(* Logix 5000 project; controller WP_Ottawa_Data_Concentrator_1 vendor 1 type 14 code 167 rev 32.14; software revision 32.04 *)
// Data Concentrator

TASK MainTask (continuous, watchdog 500 ms) : MainProgram, LN31

MODULES
   Local : vendor 1 type 14 code 167 (ICP 0, rev 32.14)
      Local_Network : vendor 1 type 12 code 200 (ICP 1, Ethernet 192.168.1.2, rev 11.2)
      Plant_Network : vendor 1 type 12 code 200 (ICP 2, Ethernet 10.31.12.136, rev 11.2)
         WP_Ottawa_Simulator_PLC : vendor 1 type 14 code 156 (Ethernet 10.31.12.137, rev 32.1, $a37dfcfc$ RPI 20 ms)   // WP_Ottawa_Simulator_PLC
         Upr_Line_PLC : vendor 1 type 12 code 200 (Ethernet 10.31.13.135, rev 11.2, Output RPI 10 ms)
            Upright_Line : vendor 1 type 14 code 213 (ICP 0, rev 31.1, $771d54c0$ RPI 20 ms, $aa9c0943$ RPI 20 ms, $f776f99a$ RPI 20 ms, $f5df2af5$ RPI 20 ms, $e50c8bc4$ RPI 20 ms, $a2ad16b7$ RPI 20 ms, $a4c949be$ RPI 20 ms, $f02d2109$ RPI 20 ms, $56660608$ RPI 20 ms, $0d2a626b$ RPI 20 ms, $ec5ac722$ RPI 20 ms, $27c2d75d$ RPI 20 ms, $f8c5678c$ RPI 20 ms, $9b57805f$ RPI 20 ms, $1c2d35c6$ RPI 20 ms, $a70581f1$ RPI 20 ms, $e44b9450$ RPI 20 ms, $3b304493$ RPI 20 ms, $244199aa$ RPI 20 ms, $c2e494c5$ RPI 20 ms, $b4e2b054$ RPI 20 ms, $661cc307$ RPI 20 ms, $eafc36ce$ RPI 20 ms, $ac2dc3d9$ RPI 20 ms)
END_MODULES

TYPE Barcode_SNModel :
STRUCT
   Data : STRING[5];
   Bit : BOOL[32];
END_STRUCT
END_TYPE

TYPE DateTime_Type :   // Structure for the DateTime from the Controller wallclock accessed by the GSV/SSV instruction
STRUCT
   Year : DINT;
   Month : DINT;   // The month (1 - 12)
   Day : DINT;   // The day (1 - 31)
   Hour : DINT;   // hour (0 - 23)
   Minute : DINT;   // minute (0 - 59)
   Second : DINT;   // second (0 - 59)
   Microseconds : DINT;   // (0 - 999,999)
END_STRUCT
END_TYPE

TYPE DC1_To_SIM :
STRUCT
   Status : CONNECTION_STATUS;
   Data : INT[225];
END_STRUCT
END_TYPE

TYPE Line_To_DC :
STRUCT
   Status : CONNECTION_STATUS;
   Data : INT[225];
END_STRUCT
END_TYPE

TYPE PA_WallClock_UDDT :
STRUCT
   One_Shots : BOOL[128];
   Bool : BOOL[128];
   Real : REAL[50];
   Dbl_Int : DINT[50];
   Int : INT[50];
   Pointer1 : INT;
   Pointer2 : INT;
   Pointer3 : INT;
   Pointer4 : INT;
   Pointer5 : INT;
   Timer : TIMER[50];
   Counter : COUNTER[25];
   Control : CONTROL[16];
END_STRUCT
END_TYPE

TYPE SIM_To_DC :
STRUCT
   Status : CONNECTION_STATUS;
   Data : INT[225];
END_STRUCT
END_TYPE

TYPE STRING_12 :
STRUCT
   LEN : DINT;
   DATA : SINT[12];
END_STRUCT
END_TYPE

TYPE STRING_16 :
STRUCT
   LEN : DINT;
   DATA : SINT[16];
END_STRUCT
END_TYPE

TYPE STRING_24 :
STRUCT
   LEN : DINT;
   DATA : SINT[24];
END_STRUCT
END_TYPE

TYPE STRING_4 :
STRUCT
   LEN : DINT;
   DATA : SINT[4];
END_STRUCT
END_TYPE

TYPE STRING_40 :
STRUCT
   LEN : DINT;
   DATA : SINT[40];
END_STRUCT
END_TYPE

TYPE UDT_Current_Status :
STRUCT
   Area : STRING_12;
   Line : STRING_12;
   Shift : DINT;
   _1st_Shift_Avail : BOOL;
   _1st_Shift_Active : BOOL;
   _1st_Shift_Scheduled : BOOL;
   _2nd_Shift_Avail : BOOL;
   _2nd_Shift_Active : BOOL;
   _2nd_Shift_Scheduled : BOOL;
   _3rd_Shift_Avail : BOOL;
   _3rd_Shift_Active : BOOL;
   _3rd_Shift_Scheduled : BOOL;
   DayOfWeek : STRING_16;
   DayOfWeek_Int : DINT;
   Start_Time : STRING_16;
   End_Time : STRING_16;
   _1st_Break_Time : STRING_16;
   _1st_Break_Trigger : BOOL;
   _1st_Break_Active : BOOL;
   _1st_Break_Used : BOOL;
   Lunch_Time : STRING_16;
   Lunch_Trigger : BOOL;
   Lunch_Active : BOOL;
   Lunch_Used : BOOL;
   _2nd_Break_Time : STRING_16;
   _2nd_Break_Trigger : BOOL;
   _2nd_Break_Active : BOOL;
   _2nd_Break_Used : BOOL;
   Rotate_Active : BOOL;
   Rotate_Cmd : BOOL;   // 30 Second Downtime Event to Rotate the Crew
   Scheduled_Units : DINT;
   Line_Rate : DINT;   // Seconds to Construct a Component
   Line_Rate_SP : REAL;
   Units_Remaining : DINT;
   Units_Produced : DINT;
   Units_Scrapped : DINT;
   Units_Lossed : DINT;
   AY_Percent : REAL;
   Shift_Minutes_Remainng : DINT;
   Shift_Seconds_Remaining : DINT;
   DownTime_Code : DINT;
   Flex_Cmd : BOOL;
   Flex_Active : BOOL;
   FlexTo_Line : STRING_16;
   Flex_EndCmd : BOOL;
   Rotate_LEN : REAL;   // seconds
   Brk_LEN : REAL;   // minutes
   Lunch_LEN : REAL;   // minutes
   Break_Stop_On : BOOL;
   Break_Stop_Allowed : BOOL;
   Flex_Stop_On : BOOL;
   Flex_Stop_Allowed : BOOL;
   Rotate_Stop_On : BOOL;
   Rotate_Stop_Allowed : BOOL;
   S1_Scheduled : DINT;
   S2_Scheduled : DINT;
   S3_Scheduled : DINT;
   Shift_Scheduled : BOOL;
   Shift_Active : BOOL;
   RateToMakeSchedule : REAL;
   Theoretical_Units : DINT;
   Standard_LineRate : REAL;
   Running : BOOL;
   State : DINT;
   LineWide_Event : DINT;
   Units_Rejected : DINT;
END_STRUCT
END_TYPE

TYPE UDT_Daily_Schedule :
STRUCT
   _1st_Shift_Avail : BOOL;
   _1st_Shift_Start : STRING_16;
   _1st_Shift_End : STRING_16;
   _1st_Shift_Break1_Start : STRING_16;
   _1st_Shift_Break1_Length : DINT;   // Minutes
   _1st_Shift_Lunch_Start : STRING_16;
   _1st_Shift_Lunch_Length : DINT;   // Minutes
   _1st_Shift_Break2_Start : STRING_16;
   _1st_Shift_Break2_Length : DINT;   // Minutes
   _2nd_Shift_Avail : BOOL;
   _2nd_Shift_Start : STRING_16;
   _2nd_Shift_End : STRING_16;
   _2nd_Shift_Break1_Start : STRING_16;
   _2nd_Shift_Break1_Length : DINT;   // Minutes
   _2nd_Shift_Lunch_Start : STRING_16;
   _2nd_Shift_Lunch_Length : DINT;   // Minutes
   _2nd_Shift_Break2_Start : STRING_16;
   _2nd_Shift_Break2_Length : DINT;   // Minutes
   _3rd_Shift_Avail : BOOL;
   _3rd_Shift_Start : STRING_16;
   _3rd_Shift_End : STRING_16;
   _3rd_Shift_Break1_Start : STRING_16;
   _3rd_Shift_Break1_Length : DINT;   // Minutes
   _3rd_Shift_Lunch_Start : STRING_16;
   _3rd_Shift_Lunch_Length : DINT;   // Minutes
   _3rd_Shift_Break2_Start : STRING_16;
   _3rd_Shift_Break2_Length : DINT;   // Minutes
   Rotate_Length : DINT;   // Seconds
   Break_Stop_On : BOOL;
   Break_Stop_Allowed : BOOL;
   Flex_Stop_On : BOOL;
   Flex_Stop_Allowed : BOOL;
   Rotate_Stop_On : BOOL;
   Rotate_Stop_Allowed : BOOL;
   S1_Scheduled : DINT;
   S2_Scheduled : DINT;
   S3_Scheduled : DINT;
   RateToMakeSchedule : REAL;
END_STRUCT
END_TYPE

TYPE UDT_ShiftString_Breakdown :
STRUCT
   s1StartHour : STRING_4;
   s1StartMin : STRING_4;
   s1EndHour : STRING_4;
   s1_EndMin : STRING_4;
   s2StartHour : STRING_4;
   s2StartMin : STRING_4;
   s2EndHour : STRING_4;
   s2EndMin : STRING_4;
   s3StartHour : STRING_4;
   s3StartMin : STRING_4;
   s3EndHour : STRING_4;
   s3EndMin : STRING_4;
   break1StartHour : STRING_4;
   break1StartMin : STRING_4;
   break2StartHour : STRING_4;
   break2StartMin : STRING_4;
   lunchStartHour : STRING_4;
   lunchStartMin : STRING_4;
END_STRUCT
END_TYPE

TYPE UDT_Weekly_Schedule :
STRUCT
   Monday : UDT_Daily_Schedule;
   Tuesday : UDT_Daily_Schedule;
   Wednesday : UDT_Daily_Schedule;
   Thursday : UDT_Daily_Schedule;
   Friday : UDT_Daily_Schedule;
   Saturday : UDT_Daily_Schedule;
   Sunday : UDT_Daily_Schedule;
END_STRUCT
END_TYPE

VAR_GLOBAL   (* controller tags *)
   ay : REAL := 0.96875;
   clock_current_string : STRING[13] := ([0] := '2023', [1] := '5', [2] := '15', [3] := '14', [4] := '19', [5] := '15');
   Clock_Min_Pulse : BOOL;
   Clock_Set_Routine : PA_WallClock_UDDT := (Dbl_Int[40] := 2023, Dbl_Int[41] := 5, Dbl_Int[42] := 15, Dbl_Int[43] := 14, Dbl_Int[44] := 19, Dbl_Int[45] := 15, Dbl_Int[46] := 696501);
   DateTime_Update : BOOL;
   DayOfWeek : DINT := 1;
   DC1_clock_sync : DINT[10] := ([0] := 2023, [1] := 5, [2] := 15, [3] := 14, [4] := 19, [5] := 12);
   DC1_OPCFault : BOOL := 1;
   DC1_OPCWatchDog : BOOL;
   DC1_To_Line31SIM : DC1_To_SIM := (Status.RunMode := 1, Data[2] := 16); {produced}
   DC1_to_LN31_Messages : DINT[120] := ([2] := 1, [3] := 620, [5] := 20, [6] := 3, [7] := 20, [8] := 3, [9] := 20, [10] := 3, [11] := 20, [12] := 3, [13] := 20, [14] := 3, [15] := 20, [16] := 3, [19] := 1); {produced}
        [10]   // CURRENT SCHEDULE SHIFT 2 START MINUTE
        [11]   // CURRENT SCHEDULE SHIFT 2 END HOUR
        [12]   // CURRENT SCHEDULE SHIFT 2 END MINUTE
        [13]   // CURRENT SCHEDULE SHIFT 3 START HOUR
        [14]   // CURRENT SCHEDULE SHIFT 3 START MINUTE
        [15]   // CURRENT SCHEDULE SHIFT 3 END HOUR
        [16]   // CURRENT SCHEDULE SHIFT 3 END MINUTE
        [19].0   // SHIFT SCHEDULED
        [19].1   // OPC COMMS OKAY
        [19].2   // Shift Reset Timer Complete
        [2]   // ACTIVE SHIFT
        [3]   // Scheduled Units
        [5]   // CURRENT SCHEDULE SHIFT 1 START HOUR
        [6]   // CURRENT SCHEDULE SHIFT 1 START MINUTE
        [7]   // CURRENT SCHEDULE SHIFT 1 END HOUR
        [8]   // CURRENT SCHEDULE SHIFT 1 END MINUTE
        [9]   // CURRENT SCHEDULE SHIFT 2 START HOUR
   fifi_unload : DINT;
   IGN_DateTime_Record_Current : STRING := '2022,09,15,08:55:00';
   IGN_Day : DINT := 15;
   IGN_DayPrev : DINT := 15;
   IGN_DayString : STRING := '15';
   IGN_Hour : DINT := 14;
   IGN_HourString : STRING := '14';
   IGN_Minute : DINT := 19;
   IGN_MinuteString : STRING := '19';
   IGN_Month : DINT := 5;
   IGN_MonthString : STRING := '5';
   IGN_Second : DINT := 10;
   IGN_SecondString : STRING := '12';
   IGN_Year : DINT := 2023;
   IGN_YearString : STRING := '2023';
   Line31SIM_To_DC1 : SIM_To_DC := (Status.RunMode := 1, Data[0] := 12);
   LN31_1st_Station_Break_Code : DINT := 16;
   LN31_Assembly_MNT : DINT;
   LN31_Blocked_At_Run_Test_Exit : DINT;
   LN31_Blocked_By_Penske_CAL : DINT;
   LN31_Blocked_By_Repair : DINT;
   LN31_Blocked_By_Wrapper : DINT;
   LN31_BrazingArea_MNT : DINT;
   LN31_Charge_MNT : DINT;
   LN31_CompressorInstall_MNT : DINT;
   LN31_Current_Shift_Duration_Mins : DINT := 505;
   LN31_Current_Shift_Duration_wBreaks_Mins : DINT := 455;
   LN31_DC_Controlled_Theoretical_Units : BOOL := 1;
   LN31_DowntimeCodesMachineA : DINT[120];
   LN31_DowntimeCodesMachineB : DINT[120];
   LN31_DowntimeCodesMachineC : DINT[120];
   LN31_DowntimeCodesMachineD : DINT[120];
   LN31_DowntimeCodesMachineE : DINT[120];
   LN31_DowntimeCodesMachineF : DINT[120];
   LN31_DowntimeCodesMachineG : DINT[120];
   LN31_DowntimeCodesMachineH : DINT[120];
   LN31_DowntimeCodesMachineI : DINT[120];
   LN31_DowntimeCodesMachineOA : DINT[120];
        [9].0   // LN31 Line Running
        [9].1   // LN31 On Break or Not Scheduled
   LN31_DowntimeCodesMachineX : DINT[120];
   LN31_EStop_HMI1 : DINT;
   LN31_EStop_HMI2 : DINT;
   LN31_EStop_Main_Panel : DINT;
   LN31_EStop_Remote_Panel : DINT;
   LN31_EvacLoop_MNT : DINT;
   LN31_FPY : REAL := 88.08;
   LN31_Ignition_NewSNModel : BOOL[32];
   LN31_Ignition_SNModelMSG : STRING[5] := ([0] := 'WZF34X18DW 07', [1] := 'UC2001942');
   LN31_InspectionAndTest_MNT : DINT;
   LN31_Kit_Zone_1_Exit_Fault : DINT;
   LN31_Kitting_MNT : DINT;
   LN31_Label_Machines_Faulted : DINT;
   LN31_Label_Missing : DINT;
   LN31_MachineOverAll_MNT : DINT;
   LN31_Messages_Barcode_SNModel : Barcode_SNModel := (Data[0] := 'WZF34X18DW 07', Data[1] := 'UC2001942');
   LN31_Miscellaneous_MNT : DINT;
   LN31_MLC_Downtime : BOOL;
   LN31_Packout_MNT : DINT;
   LN31_PrefoamGlueAndFoam_MNT : DINT;
   LN31_Schedule : UDT_Current_Status := (Line := 'LN31', Shift := 1, _1st_Shift_Avail := 1, _1st_Shift_Active := 1, _1st_Shift_Scheduled := 1, _3rd_Shift_Scheduled := 1, DayOfWeek := 'Mon', DayOfWeek_Int := 1, Start_Time := '2023-05-15 07:05', End_Time := '2023-05-15 15:30', _1st_Break_Time := '09:10', Lunch_Time := '12:10', _2nd_Break_Time := '20:30', Scheduled_Units := 620, Line_Rate := 56, Units_Remaining := 415, Units_Produced := 411, Units_Lossed := 13, AY_Percent := 96.875, Break_Stop_Allowed := 1, Shift_Scheduled := 1, Shift_Active := 1, Theoretical_Units := 522, Running := 1, State := 3, Units_Rejected := 49);
        .Units_Lossed   // LN31 Rejected Count
   LN31_Schedule_Cycle_Timer : TIMER := (PRE := 44032, ACC := 751, EN := 1, TT := 1);
   LN31_Schedule_Max_Break_Duration : DINT := 50;
   LN31_Schedule_Max_Break_Timer : TIMER := (PRE := 3000000, ACC := 3000000, EN := 1, DN := 1);
   LN31_Schedule_TAKT : REAL := 44032.258;
   LN31_Scheduled_Units_Buffer : DINT := 620;
   LN31_ScheduleUnits_Produced_from_line : DINT := 412;
   LN31_Starved_By_Surge : DINT;
   LN31_Surge_Gate_Open : DINT;
   LN31_Theoretical_Units_Counter : COUNTER := (PRE := 999999, ACC := 522);
   LN31_Theoretical_Units_Counter_ONS : BOOL;
   LN31_to_DC01_Main_Messages : Line_To_DC := (Status.RunMode := 1, Data[4] := 543, Data[6] := 44, Data[9] := 1, Data[15] := 8637, Data[18] := 618, Data[19] := 74);
   LN31_Toggle_CountSource : BOOL;
   LN31_Weekly_Schedule : UDT_Weekly_Schedule := (Monday._1st_Shift_Avail := 1, Monday._1st_Shift_Start := '2023-05-15 07:05', Monday._1st_Shift_End := '2023-05-15 15:30', Monday._1st_Shift_Break1_Start := '09:10', Monday._1st_Shift_Break1_Length := 15, Monday._1st_Shift_Lunch_Start := '12:10', Monday._1st_Shift_Lunch_Length := 30, Monday._1st_Shift_Break2_Start := '20:30', Monday._1st_Shift_Break2_Length := 15, Monday._2nd_Shift_Start := '2023-05-15 20:25', Monday._2nd_Shift_End := '2023-05-15 20:30', Monday._2nd_Shift_Break1_Start := '17:45', Monday._2nd_Shift_Break1_Length := 15, Monday._2nd_Shift_Lunch_Start := '20:30', Monday._2nd_Shift_Lunch_Length := 30, Monday._2nd_Shift_Break2_Start := '12:10', Monday._2nd_Shift_Break2_Length := 15, Monday._3rd_Shift_Avail := 1, Monday._3rd_Shift_Start := '2023-05-14 21:35', Monday._3rd_Shift_End := '2023-05-15 06:00', Monday._3rd_Shift_Break1_Start := '01:00', Monday._3rd_Shift_Break1_Length := 15, Monday._3rd_Shift_Lunch_Start := '03:00', Monday._3rd_Shift_Lunch_Length := 30, Monday._3rd_Shift_Break2_Start := '04:00', Monday._3rd_Shift_Break2_Length := 15, Monday.S1_Scheduled := 620, Monday.S3_Scheduled := 620, Tuesday._1st_Shift_Avail := 1, Tuesday._1st_Shift_Start := '2023-05-16 07:05', Tuesday._1st_Shift_End := '2023-05-16 15:30', Tuesday._1st_Shift_Break1_Start := '09:10', Tuesday._1st_Shift_Break1_Length := 15, Tuesday._1st_Shift_Lunch_Start := '12:10', Tuesday._1st_Shift_Lunch_Length := 30, Tuesday._1st_Shift_Break2_Start := '20:30', Tuesday._1st_Shift_Break2_Length := 15, Tuesday._2nd_Shift_Start := '2023-05-16 20:25', Tuesday._2nd_Shift_End := '2023-05-16 20:30', Tuesday._2nd_Shift_Break1_Start := '17:45', Tuesday._2nd_Shift_Break1_Length := 15, Tuesday._2nd_Shift_Lunch_Start := '20:30', Tuesday._2nd_Shift_Lunch_Length := 30, Tuesday._2nd_Shift_Break2_Start := '12:10', Tuesday._2nd_Shift_Break2_Length := 15, Tuesday._3rd_Shift_Avail := 1, Tuesday._3rd_Shift_Start := '2023-05-15 21:35', Tuesday._3rd_Shift_End := '2023-05-16 06:00', Tuesday._3rd_Shift_Break1_Start := '1:00', Tuesday._3rd_Shift_Break1_Length := 15, Tuesday._3rd_Shift_Lunch_Start := '03:00', Tuesday._3rd_Shift_Lunch_Length := 30, Tuesday._3rd_Shift_Break2_Start := '04:00', Tuesday._3rd_Shift_Break2_Length := 15, Tuesday.S1_Scheduled := 620, Tuesday.S3_Scheduled := 620, Wednesday._1st_Shift_Avail := 1, Wednesday._1st_Shift_Start := '2023-05-17 07:05', Wednesday._1st_Shift_End := '2023-05-17 15:30', Wednesday._1st_Shift_Break1_Start := '09:10',
        Wednesday._1st_Shift_Break1_Length := 15, Wednesday._1st_Shift_Lunch_Start := '12:10', Wednesday._1st_Shift_Lunch_Length := 30, Wednesday._1st_Shift_Break2_Start := '20:30', Wednesday._1st_Shift_Break2_Length := 15, Wednesday._2nd_Shift_Start := '2023-05-17 20:25', Wednesday._2nd_Shift_End := '2023-05-17 20:30', Wednesday._2nd_Shift_Break1_Start := '17:45', Wednesday._2nd_Shift_Break1_Length := 15, Wednesday._2nd_Shift_Lunch_Start := '20:30', Wednesday._2nd_Shift_Lunch_Length := 30, Wednesday._2nd_Shift_Break2_Start := '12:10', Wednesday._2nd_Shift_Break2_Length := 15, Wednesday._3rd_Shift_Avail := 1, Wednesday._3rd_Shift_Start := '2023-05-16 21:35', Wednesday._3rd_Shift_End := '2023-05-17 06:00', Wednesday._3rd_Shift_Break1_Start := '01:00', Wednesday._3rd_Shift_Break1_Length := 15, Wednesday._3rd_Shift_Lunch_Start := '03:00', Wednesday._3rd_Shift_Lunch_Length := 30, Wednesday._3rd_Shift_Break2_Start := '04:00', Wednesday._3rd_Shift_Break2_Length := 15, Wednesday.S1_Scheduled := 620, Wednesday.S3_Scheduled := 620, Thursday._1st_Shift_Avail := 1, Thursday._1st_Shift_Start := '2023-05-18 07:05', Thursday._1st_Shift_End := '2023-05-18 15:30', Thursday._1st_Shift_Break1_Start := '09:10', Thursday._1st_Shift_Break1_Length := 15, Thursday._1st_Shift_Lunch_Start := '12:10', Thursday._1st_Shift_Lunch_Length := 30, Thursday._1st_Shift_Break2_Start := '20:30', Thursday._1st_Shift_Break2_Length := 15, Thursday._2nd_Shift_Start := '2023-05-18 20:25', Thursday._2nd_Shift_End := '2023-05-18 20:30', Thursday._2nd_Shift_Break1_Start := '17:45', Thursday._2nd_Shift_Break1_Length := 15, Thursday._2nd_Shift_Lunch_Start := '20:30', Thursday._2nd_Shift_Lunch_Length := 30, Thursday._2nd_Shift_Break2_Start := '12:10', Thursday._2nd_Shift_Break2_Length := 15, Thursday._3rd_Shift_Avail := 1, Thursday._3rd_Shift_Start := '2023-05-17 21:35', Thursday._3rd_Shift_End := '2023-05-18 06:00', Thursday._3rd_Shift_Break1_Start := '01:00', Thursday._3rd_Shift_Break1_Length := 15, Thursday._3rd_Shift_Lunch_Start := '03:00', Thursday._3rd_Shift_Lunch_Length := 30, Thursday._3rd_Shift_Break2_Start := '04:00', Thursday._3rd_Shift_Break2_Length := 15, Thursday.S1_Scheduled := 620, Thursday.S3_Scheduled := 620, Friday._1st_Shift_Avail := 1, Friday._1st_Shift_Start := '2023-05-19 07:05', Friday._1st_Shift_End := '2023-05-19 15:30', Friday._1st_Shift_Break1_Start := '09:10', Friday._1st_Shift_Break1_Length := 15, Friday._1st_Shift_Lunch_Start := '12:10', Friday._1st_Shift_Lunch_Length := 30, Friday._1st_Shift_Break2_Start := '20:30',
        Friday._1st_Shift_Break2_Length := 15, Friday._2nd_Shift_Start := '2023-05-19 20:25', Friday._2nd_Shift_End := '2023-05-19 20:30', Friday._2nd_Shift_Break1_Start := '17:45', Friday._2nd_Shift_Break1_Length := 15, Friday._2nd_Shift_Lunch_Start := '20:30', Friday._2nd_Shift_Lunch_Length := 30, Friday._2nd_Shift_Break2_Start := '12:10', Friday._2nd_Shift_Break2_Length := 15, Friday._3rd_Shift_Avail := 1, Friday._3rd_Shift_Start := '2023-05-18 21:35', Friday._3rd_Shift_End := '2023-05-19 06:00', Friday._3rd_Shift_Break1_Start := '01:00', Friday._3rd_Shift_Break1_Length := 15, Friday._3rd_Shift_Lunch_Start := '03:00', Friday._3rd_Shift_Lunch_Length := 30, Friday._3rd_Shift_Break2_Start := '04:00', Friday._3rd_Shift_Break2_Length := 15, Friday.S1_Scheduled := 620, Friday.S3_Scheduled := 620, Saturday._1st_Shift_Start := '2023-05-20 07:05', Saturday._1st_Shift_End := '2023-05-20 16:30', Saturday._1st_Shift_Break1_Start := '09:10', Saturday._1st_Shift_Break1_Length := 15, Saturday._1st_Shift_Lunch_Start := '12:10', Saturday._1st_Shift_Lunch_Length := 30, Saturday._1st_Shift_Break2_Start := '18:45', Saturday._1st_Shift_Break2_Length := 15, Saturday._2nd_Shift_Start := '2023-05-20 17:00', Saturday._2nd_Shift_End := '2023-05-20 17:01', Saturday._2nd_Shift_Break1_Start := '17:45', Saturday._2nd_Shift_Break1_Length := 15, Saturday._2nd_Shift_Lunch_Start := '20:30', Saturday._2nd_Shift_Lunch_Length := 30, Saturday._2nd_Shift_Break2_Start := '12:10', Saturday._2nd_Shift_Break2_Length := 15, Saturday._3rd_Shift_Start := '2023-05-19 20:35', Saturday._3rd_Shift_End := '2023-05-20 06:00', Saturday._3rd_Shift_Break1_Start := '01:00', Saturday._3rd_Shift_Break1_Length := 15, Saturday._3rd_Shift_Lunch_Start := '03:00', Saturday._3rd_Shift_Lunch_Length := 30, Saturday._3rd_Shift_Break2_Start := '05:00', Saturday._3rd_Shift_Break2_Length := 15, Sunday._1st_Shift_Start := '2023-05-21 07:05', Sunday._1st_Shift_End := '2023-05-21 16:30', Sunday._1st_Shift_Break1_Start := '09:0', Sunday._1st_Shift_Break1_Length := 15, Sunday._1st_Shift_Lunch_Start := '12:10', Sunday._1st_Shift_Lunch_Length := 30, Sunday._1st_Shift_Break2_Start := '18:45', Sunday._1st_Shift_Break2_Length := 15, Sunday._2nd_Shift_Start := '2023-05-21 17:00', Sunday._2nd_Shift_End := '2023-05-21 17:01', Sunday._2nd_Shift_Break1_Start := '17:45', Sunday._2nd_Shift_Break1_Length := 30, Sunday._2nd_Shift_Lunch_Start := '20:30', Sunday._2nd_Shift_Lunch_Length := 30, Sunday._2nd_Shift_Break2_Start := '12:10', Sunday._2nd_Shift_Break2_Length := 15,
        Sunday._3rd_Shift_Start := '2023-05-20 20:35', Sunday._3rd_Shift_End := '2023-05-21 06:00', Sunday._3rd_Shift_Break1_Start := '01:00', Sunday._3rd_Shift_Break1_Length := 140, Sunday._3rd_Shift_Lunch_Start := '03:00', Sunday._3rd_Shift_Lunch_Length := 30, Sunday._3rd_Shift_Break2_Start := '05:00', Sunday._3rd_Shift_Break2_Length := 10);
   LN31_WorkstationsA : DINT[120];
   LN31_WorkstationsB : DINT[120] := ([3] := 1048592);
   LN31_WorkstationsC : DINT[120];
   LN31_WorkstationsD : DINT[120];
   LN31_WorkstationsE : DINT[120];
   LN31_WorkstationsF : DINT[120];
   LN31_WorkstationsG : DINT[120];
   LN31_WorkstationsH : DINT[120];
   LN31_WorkstationsI : DINT[120];
   LN31_WorkstationsOA : DINT[120] := ([4] := 411, [6] := 56, [9] := 1, [15] := 8808, [16] := 49, [17] := 1, [18] := 410);
        [15]   // LN31 Lodestar FPY Decimal as Integer
        [17]   // LN31 Active Shift
        [18]   // LN31 Scheduled Units (Run Target Count)
        [19]   // LN31 Lost Unit Count ( Reject Count)
        [20]   // LN31 Main Line Active DT Code
        [21]   // LN31 Sub Process 1 Machine DT Code
        [22]   // LN31 Sub Process 2 Machine DT Code
        [23]   // LN31 Sub Process 3 Machine DT Code
        [24]   // LN31 Sub Process 4 Machine DT Code
        [25]   // LN31 Sub Process 5 Machine DT Code
        [26]   // LN31 Sub Process 6 Machine DT Code
        [27]   // LN31 Sub Process 7 Machine DT Code
        [28]   // LN31 Sub Process 8 Machine DT Code
        [29]   // LN31 Sub Process 9 Machine DT Code
        [30]   // LN31 Sub Process 10 Machine DT Code
        [4]   // LN31 Actual Unit Count (Lodestar Crated)
        [6]   // LN31 Takt Target Time
        [9].0   // Line Running
        [9].1   // On Break or Not Scheduled
   LN31_WorkstationsX : DINT[120] := ([7] := 1048592, [8] := 1048592, [9] := 1048592, [10] := 1048592, [11] := 1048592, [12] := 1048592);
   LN31_Wrong_Compressor : DINT;
   LN31_Z22F_Over_Cycle_Time : DINT;
   LN31EAM02 : DINT;
   LN31EAM03 : DINT;
   LN31EFM01 : DINT;
   LN31EFM02 : DINT;
   LN31EFM03 : DINT;
   LN31EGM01 : DINT;
   LN31EGM02 : DINT;
   LN31EGM03 : DINT;
   LN31EGM04 : DINT;
   LN31EHS01 : DINT;
   LN31EHS02 : DINT;
   LN31EHS03 : DINT;
   LN31EHS04 : DINT;
   LN31EHS05 : DINT;
   LN31EHS06 : DINT;
   LN31EHS07 : DINT;
   LN31EHS08 : DINT;
   LN31EIS05 : DINT;
   LN31NCM02 : DINT;
   LN31NDM01 : DINT;
   LN31NDM02 : DINT;
   LN31NDM03 : DINT;
   LN31NIS02 : DINT;
   LN31NIS03 : DINT;
   LN31NIS04 : DINT;
   LN31NIS06 : DINT;
   LN31NIS07 : DINT;
   LN31NIS08 : DINT;
   LN31NIS09 : DINT;
   LN31NIS10 : DINT;
   LN31NIS11 : DINT;
   LN31NIS12 : DINT;
   LN31NIS13 : DINT;
   LN31NIS14 : DINT;
   LN31NIS15 : DINT;
   LN31NIS16 : DINT;
   LN31NIS17 : DINT;
   LN31SBM01 : DINT;
   LN31SBM02 : DINT;
   LN31SBM03 : DINT;
   LN31SBM04 : DINT;
   LN31SBM05 : DINT;
   LN31SCM01 : DINT;
   LN31SDM03 : DINT;
   LN31SIS02 : DINT;
   LN31SIS06 : DINT;
   LN31WAM01 : DINT;
   LN31WAM02 : DINT;
   LN31WEM01 : DINT;
   LN31WEM02 : DINT;
   LN31WEM03 : DINT;
   LN31WEM04 : DINT;
   LN31WEM05 : DINT;
   LN31WEM06 : DINT;
   LN31WEM07 : DINT;
   LN31WEM08 : DINT;
   LN31WEM09 : DINT;
   LN31WFM01 : DINT;
   LN31WFM02 : DINT;
   LN31WFM03 : DINT;
   LN31WGM02 : DINT;
   LN31WGM04 : DINT;
   LN31WIS01 : DINT;
   LN31XAM01 : DINT;
   LN31XAM02 : DINT;
   LN31XAS01 : DINT;
   LN31XAS02 : DINT;
   LN31XBM01 : DINT;
   LN31XBM02 : DINT;
   LN31XBS01 : DINT;
   LN31XBS02 : DINT;
   LN31XCM01 : DINT;
   LN31XCM02 : DINT;
   LN31XCS01 : DINT;
   LN31XCS02 : DINT;
   LN31XDM01 : DINT;
   LN31XDM02 : DINT;
   LN31XDS01 : DINT;
   LN31XDS02 : DINT;
   LN31XEM01 : DINT;
   LN31XEM02 : DINT;
   LN31XES01 : DINT;
   LN31XES02 : DINT;
   LN31XFM01 : DINT;
   LN31XFM02 : DINT;
   LN31XFS01 : DINT;
   LN31XFS02 : DINT;
   LN31XGM01 : DINT;
   LN31XGM02 : DINT;
   LN31XGS01 : DINT;
   LN31XGS02 : DINT;
   LN31XHM01 : DINT;
   LN31XHM02 : DINT;
   LN31XHS01 : DINT;
   LN31XHS02 : DINT;
   LN31XIM01 : DINT;
   LN31XIM02 : DINT;
   LN31XIM03 : DINT;
   LN31XIS01 : DINT;
   LN31XIS02 : DINT;
   LN31XIS03 : DINT;
   local : TIMER := (PRE := 2000, ACC := 1827, EN := 1, TT := 1);
   null : STRING;
   NULL_String : STRING;
   Previous_Shift_Count : DINT := 463;
   scc : CONTROL := (LEN := 60, POS := 59);   // Shift Count History
   Shift_count_history : DINT[62];
   Shift_reset_timer : TIMER := (PRE := 2000);
   Test : MESSAGE;
        MessageParameters(ServiceCode := 16#004c, LocalElement := Test1, ...)
   Test1 : DINT;
   Test_Result : DINT := 1;
   TestDateTime : DINT;
   THEORETICAL_TEST : BOOL;
END_VAR

PROGRAM LN31   (* main routine MainRoutine *)
VAR
   Average_Array : DINT[20] := ([0] := 30000, [1] := 30000, [2] := 30000, [3] := 30000, [4] := 30000, [5] := 30000, [6] := 30000, [7] := 30000, [8] := 30000, [9] := 30000);   // AVERAGE UNIT ASSEMBLY TIME (LAST 10 UNITS)
   Average_Sum : DINT := 300000;
   Averaged_LineSpeed : REAL := 30.0;
   badModel : STRING_40;
   Break1_Hour : DINT := 9;
   Break1_Hour_String : STRING_4 := '09';
   Break1_Length : DINT := 15;
   Break1_Min : DINT := 10;
   Break1_Min_String : STRING_4 := '10';
   Break2_Hour : DINT := 20;
   Break2_Hour_String : STRING_4 := '20';
   Break2_Length : DINT := 15;
   Break2_Min : DINT := 30;
   Break2_Min_String : STRING_4 := '30';
   Break_1stStation : BOOL;
   Break_LineWide : BOOL;
   Break_WorkCenter : BOOL;
   Break_Workstation : BOOL;
   CurrentSchedule : UDT_ShiftString_Breakdown := (s1StartHour := '20', s1StartMin := '3-', s1EndHour := '20', s1_EndMin := '3-', s2StartHour := '20', s2StartMin := '3-', s2EndHour := '20', s2EndMin := '3-', s3StartHour := '20', s3StartMin := '3-', s3EndHour := '20', s3EndMin := '3-');
   End_Hour : DINT := 20;
   End_Hour_String : STRING_4 := '20';
   End_Min : DINT := 3;
   End_Min_String : STRING_4 := '3-';
   firstCharacter : STRING_40 := 'W';
   Local_Timer : TIMER[10] := ([0].PRE := 30000, [0].ACC := 30000, [0].EN := 1, [0].DN := 1, [1].PRE := 4000, [1].ACC := 4000, [1].EN := 1, [1].DN := 1, [2].PRE := 8000, [3].PRE := 2000, [3].ACC := 1538, [3].EN := 1, [3].TT := 1, [4].PRE := 280, [4].ACC := 95, [4].EN := 1, [4].TT := 1);
        [0]   // UNIT ASSEMBLY TIMER
        [1]   // BARCODE TRANSFER TO LODESTAR TRIGGER TIMER
        [2]   // BARCOE TRANFER TO LODESTAR SECOND CHANCE TIMER
        [3]   // LINE PLC WRITE MESSAGE INSTRUCTION TIMER
        [4]   // LINE PLC READ MESSAGE INSTRUCTION TIMER
   Lunch_Hour : DINT := 12;
   Lunch_Hour_String : STRING_4 := '12';
   Lunch_Length : DINT := 30;
   Lunch_Min : DINT := 10;
   Lunch_Min_String : STRING_4 := '10';
   msg192_reset_timer : TIMER := (PRE := 3000);
   ONS_20 : DINT := 3;
        .0   // BARCODE READ FROM LODESTAR STATUS ONE SHOT
        .1   // CLEAR BARCODE READ FROM LODESTAR STATUS ONE SHOT
   PreviousCount : DINT := 411;
   previousSerialNumber : STRING := 'M91940611';
   PreviousShift : DINT := 1;
   readIndex : DINT := 31;
   register : DINT := 9;   // ARRAY POINTER FOR AVERAGE ASSEMBLY TIME ARRAY
   Shift_Reset : BOOL;
   Shift_Reset_ONS : BOOL := 1;
   Start_Hour : DINT := 20;
   Start_Hour_String : STRING_4 := '20';
   Start_Min : DINT := 3;
   Start_Min_String : STRING_4 := '3-';
   tempIndex : DINT := 22;
   theoreticalUnitsReal : REAL;
   writeIndex : DINT;
END_VAR

ROUTINE MainRoutine   (* ladder *)
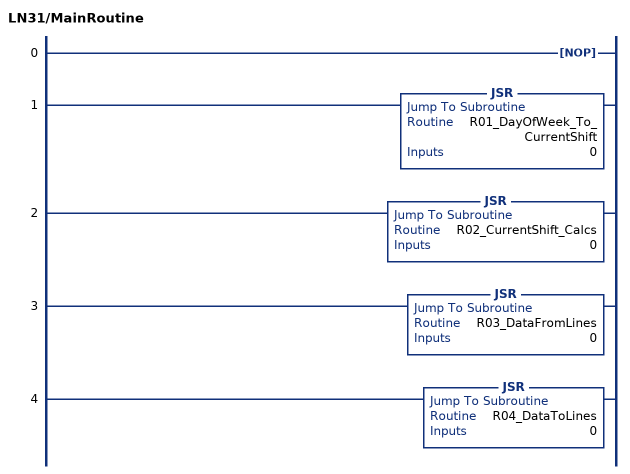
   0: NOP();
   1: JSR(R01_DayOfWeek_To_CurrentShift,0);
   2: JSR(R02_CurrentShift_Calcs,0);
   3: JSR(R03_DataFromLines,0);
   4: JSR(R04_DataToLines,0);
END_ROUTINE

ROUTINE R01_DayOfWeek_To_CurrentShift   (* ladder *)
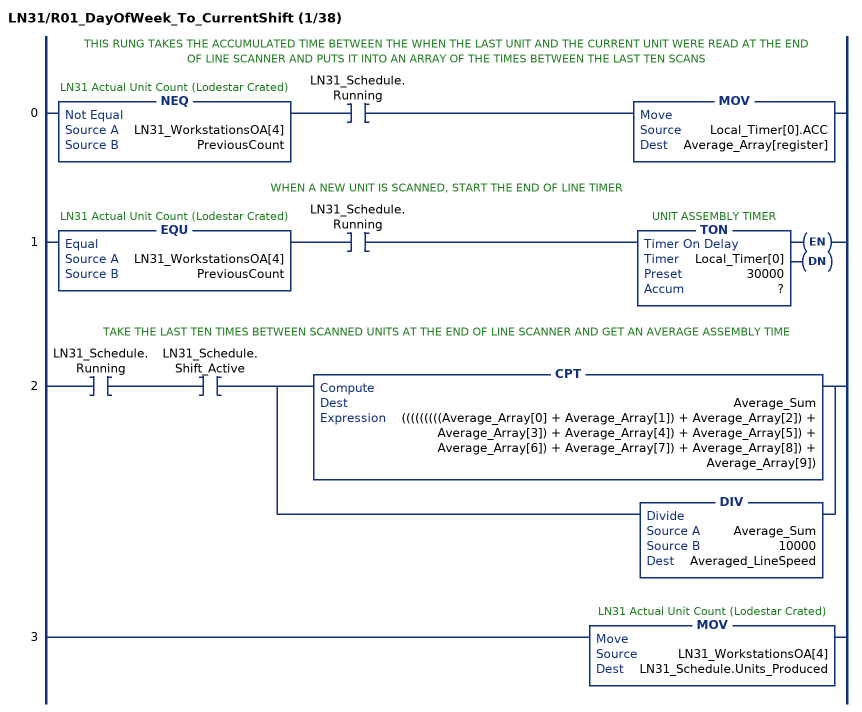
   // THIS RUNG TAKES THE ACCUMULATED TIME BETWEEN THE WHEN THE LAST UNIT AND THE CURRENT UNIT WERE READ AT THE END OF LINE SCANNER AND PUTS IT INTO AN ARRAY OF THE TIMES BETWEEN THE LAST TEN SCANS
   0: NEQ(LN31_WorkstationsOA[4],PreviousCount)XIC(LN31_Schedule.Running)MOV(Local_Timer[0].ACC,Average_Array[register]);
   // WHEN A NEW UNIT IS SCANNED, START THE END OF LINE TIMER
   1: EQU(LN31_WorkstationsOA[4],PreviousCount)XIC(LN31_Schedule.Running)TON(Local_Timer[0],?,?);
   // TAKE THE LAST TEN TIMES BETWEEN SCANNED UNITS AT THE END OF LINE SCANNER AND GET AN AVERAGE ASSEMBLY TIME
   2: XIC(LN31_Schedule.Running)XIC(LN31_Schedule.Shift_Active)[CPT(Average_Sum,(((((((((Average_Array[0] + Average_Array[1]) + Average_Array[2]) + Average_Array[3]) + Average_Array[4]) + Average_Array[5]) + Average_Array[6]) + Average_Array[7]) + Average_Array[8]) + Average_Array[9])) ,DIV(Average_Sum,10000,Averaged_LineSpeed) ];
   3: MOV(LN31_WorkstationsOA[4],LN31_Schedule.Units_Produced);
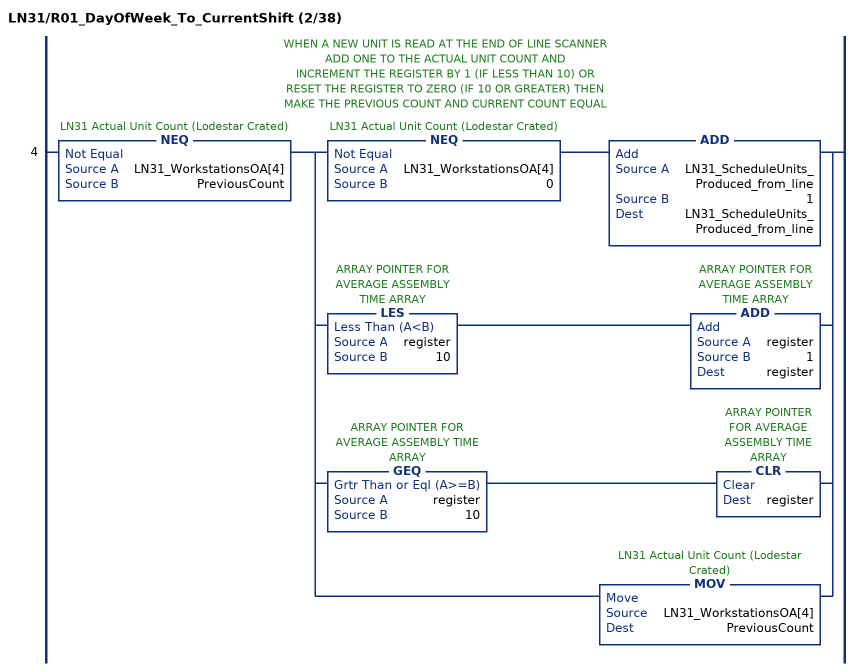
   // WHEN A NEW UNIT IS READ AT THE END OF LINE SCANNER
   // ADD ONE TO THE ACTUAL UNIT COUNT AND
   // INCREMENT THE REGISTER BY 1 (IF LESS THAN 10) OR
   // RESET THE REGISTER TO ZERO (IF 10 OR GREATER) THEN
   // MAKE THE PREVIOUS COUNT AND CURRENT COUNT EQUAL
   4: NEQ(LN31_WorkstationsOA[4],PreviousCount)[NEQ(LN31_WorkstationsOA[4],0) ADD(LN31_ScheduleUnits_Produced_from_line,1,LN31_ScheduleUnits_Produced_from_line) ,LES(register,10) ADD(register,1,register) ,GEQ(register,10) CLR(register) ,MOV(LN31_WorkstationsOA[4],PreviousCount) ];
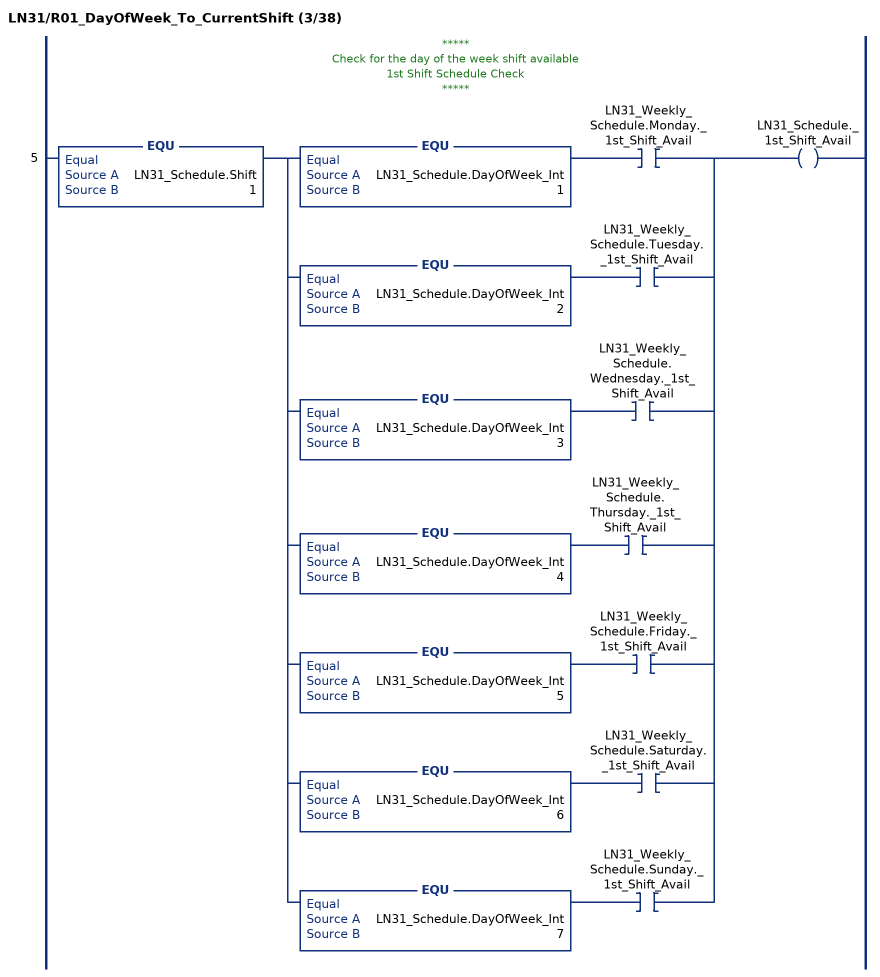
   // *****
   // Check for the day of the week shift available
   // 1st Shift Schedule Check
   // *****
   5: EQU(LN31_Schedule.Shift,1)[EQU(LN31_Schedule.DayOfWeek_Int,1) XIC(LN31_Weekly_Schedule.Monday._1st_Shift_Avail) ,EQU(LN31_Schedule.DayOfWeek_Int,2) XIC(LN31_Weekly_Schedule.Tuesday._1st_Shift_Avail) ,EQU(LN31_Schedule.DayOfWeek_Int,3) XIC(LN31_Weekly_Schedule.Wednesday._1st_Shift_Avail) ,EQU(LN31_Schedule.DayOfWeek_Int,4) XIC(LN31_Weekly_Schedule.Thursday._1st_Shift_Avail) ,EQU(LN31_Schedule.DayOfWeek_Int,5) XIC(LN31_Weekly_Schedule.Friday._1st_Shift_Avail) ,EQU(LN31_Schedule.DayOfWeek_Int,6) XIC(LN31_Weekly_Schedule.Saturday._1st_Shift_Avail) ,EQU(LN31_Schedule.DayOfWeek_Int,7) XIC(LN31_Weekly_Schedule.Sunday._1st_Shift_Avail) ]OTE(LN31_Schedule._1st_Shift_Avail);
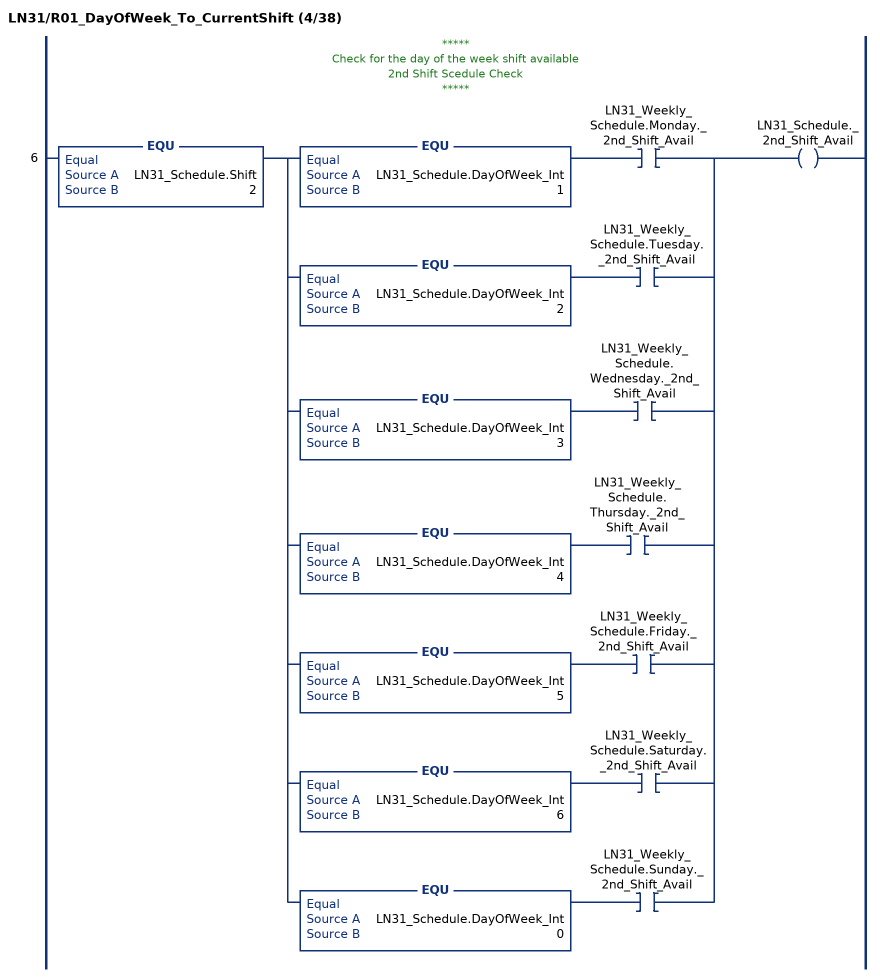
   // *****
   // Check for the day of the week shift available
   // 2nd Shift Scedule Check
   // *****
   6: EQU(LN31_Schedule.Shift,2)[EQU(LN31_Schedule.DayOfWeek_Int,1) XIC(LN31_Weekly_Schedule.Monday._2nd_Shift_Avail) ,EQU(LN31_Schedule.DayOfWeek_Int,2) XIC(LN31_Weekly_Schedule.Tuesday._2nd_Shift_Avail) ,EQU(LN31_Schedule.DayOfWeek_Int,3) XIC(LN31_Weekly_Schedule.Wednesday._2nd_Shift_Avail) ,EQU(LN31_Schedule.DayOfWeek_Int,4) XIC(LN31_Weekly_Schedule.Thursday._2nd_Shift_Avail) ,EQU(LN31_Schedule.DayOfWeek_Int,5) XIC(LN31_Weekly_Schedule.Friday._2nd_Shift_Avail) ,EQU(LN31_Schedule.DayOfWeek_Int,6) XIC(LN31_Weekly_Schedule.Saturday._2nd_Shift_Avail) ,EQU(LN31_Schedule.DayOfWeek_Int,0) XIC(LN31_Weekly_Schedule.Sunday._2nd_Shift_Avail) ]OTE(LN31_Schedule._2nd_Shift_Avail);
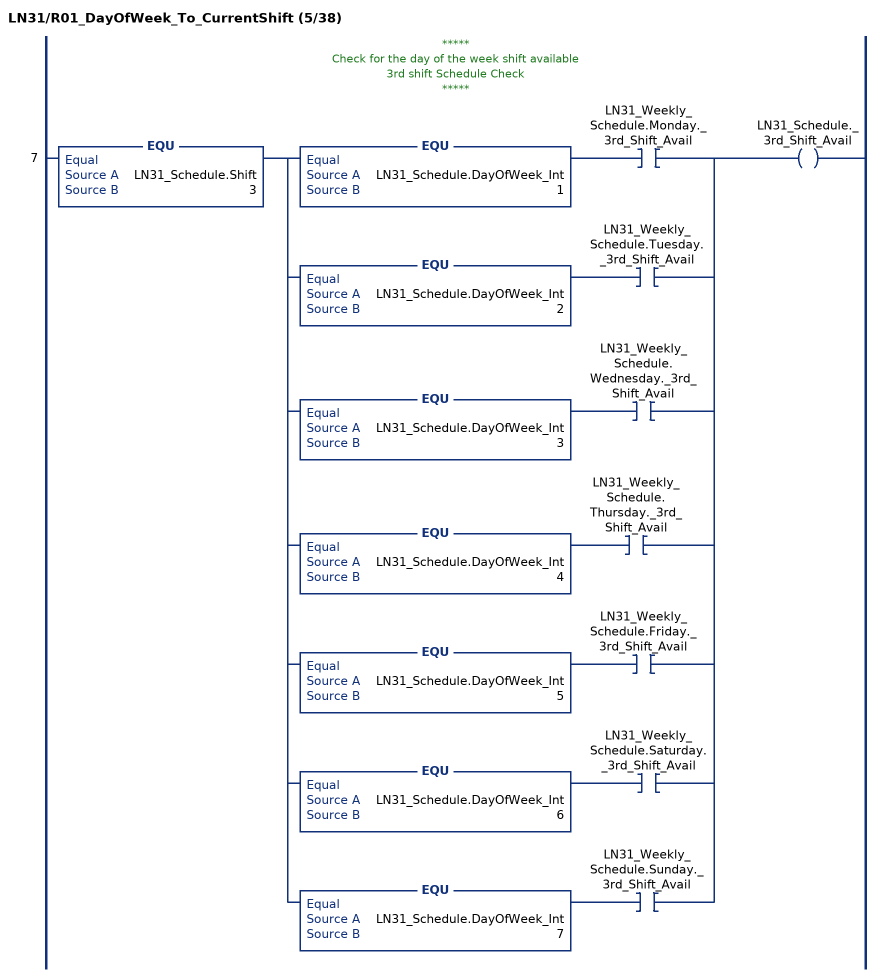
   // *****
   // Check for the day of the week shift available
   // 3rd shift Schedule Check
   // *****
   7: EQU(LN31_Schedule.Shift,3)[EQU(LN31_Schedule.DayOfWeek_Int,1) XIC(LN31_Weekly_Schedule.Monday._3rd_Shift_Avail) ,EQU(LN31_Schedule.DayOfWeek_Int,2) XIC(LN31_Weekly_Schedule.Tuesday._3rd_Shift_Avail) ,EQU(LN31_Schedule.DayOfWeek_Int,3) XIC(LN31_Weekly_Schedule.Wednesday._3rd_Shift_Avail) ,EQU(LN31_Schedule.DayOfWeek_Int,4) XIC(LN31_Weekly_Schedule.Thursday._3rd_Shift_Avail) ,EQU(LN31_Schedule.DayOfWeek_Int,5) XIC(LN31_Weekly_Schedule.Friday._3rd_Shift_Avail) ,EQU(LN31_Schedule.DayOfWeek_Int,6) XIC(LN31_Weekly_Schedule.Saturday._3rd_Shift_Avail) ,EQU(LN31_Schedule.DayOfWeek_Int,7) XIC(LN31_Weekly_Schedule.Sunday._3rd_Shift_Avail) ]OTE(LN31_Schedule._3rd_Shift_Avail);
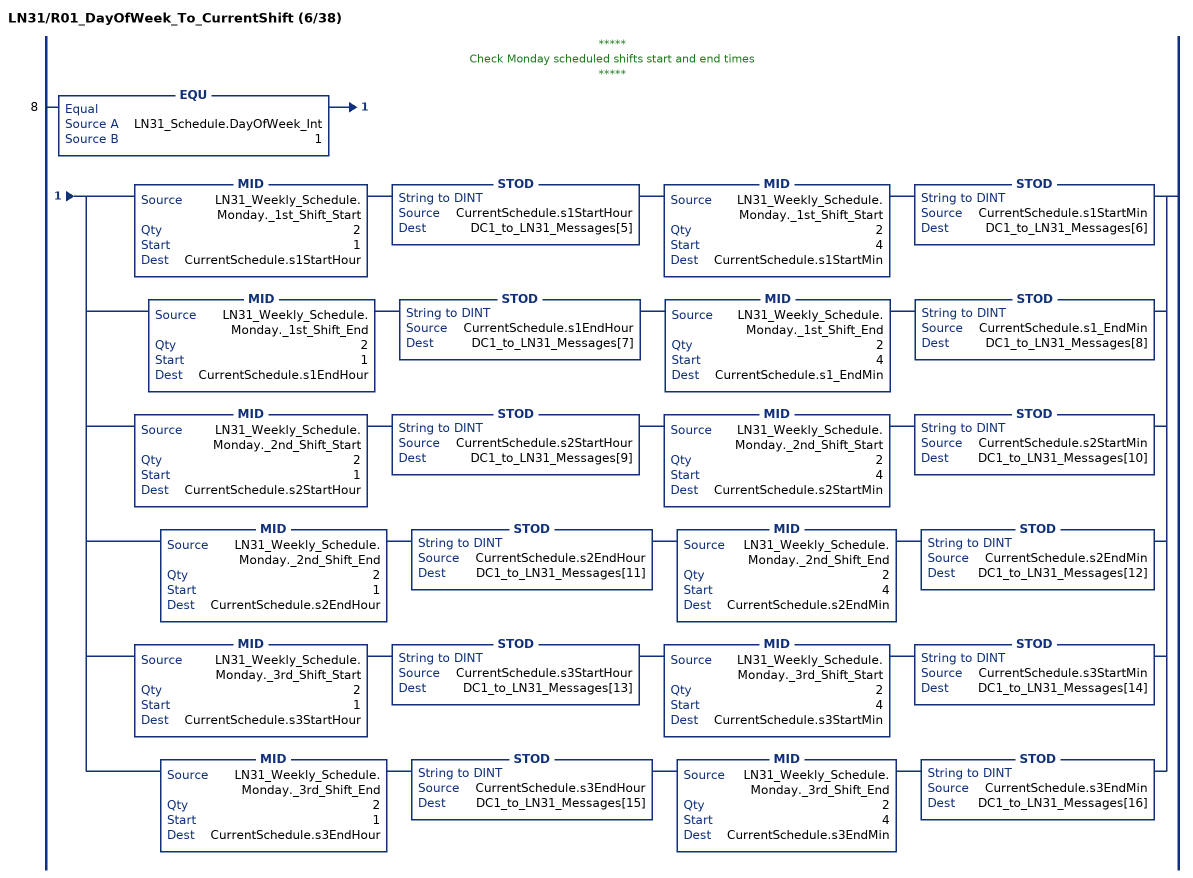
   // *****
   // Check Monday scheduled shifts start and end times
   // *****
   8: EQU(LN31_Schedule.DayOfWeek_Int,1)[MID(LN31_Weekly_Schedule.Monday._1st_Shift_Start,2,1,CurrentSchedule.s1StartHour) STOD(CurrentSchedule.s1StartHour,DC1_to_LN31_Messages[5]) MID(LN31_Weekly_Schedule.Monday._1st_Shift_Start,2,4,CurrentSchedule.s1StartMin) STOD(CurrentSchedule.s1StartMin,DC1_to_LN31_Messages[6]) ,MID(LN31_Weekly_Schedule.Monday._1st_Shift_End,2,1,CurrentSchedule.s1EndHour) STOD(CurrentSchedule.s1EndHour,DC1_to_LN31_Messages[7]) MID(LN31_Weekly_Schedule.Monday._1st_Shift_End,2,4,CurrentSchedule.s1_EndMin) STOD(CurrentSchedule.s1_EndMin,DC1_to_LN31_Messages[8]) ,MID(LN31_Weekly_Schedule.Monday._2nd_Shift_Start,2,1,CurrentSchedule.s2StartHour) STOD(CurrentSchedule.s2StartHour,DC1_to_LN31_Messages[9]) MID(LN31_Weekly_Schedule.Monday._2nd_Shift_Start,2,4,CurrentSchedule.s2StartMin) STOD(CurrentSchedule.s2StartMin,DC1_to_LN31_Messages[10]) ,MID(LN31_Weekly_Schedule.Monday._2nd_Shift_End,2,1,CurrentSchedule.s2EndHour) STOD(CurrentSchedule.s2EndHour,DC1_to_LN31_Messages[11]) MID(LN31_Weekly_Schedule.Monday._2nd_Shift_End,2,4,CurrentSchedule.s2EndMin) STOD(CurrentSchedule.s2EndMin,DC1_to_LN31_Messages[12]) ,MID(LN31_Weekly_Schedule.Monday._3rd_Shift_Start,2,1,CurrentSchedule.s3StartHour) STOD(CurrentSchedule.s3StartHour,DC1_to_LN31_Messages[13]) MID(LN31_Weekly_Schedule.Monday._3rd_Shift_Start,2,4,CurrentSchedule.s3StartMin) STOD(CurrentSchedule.s3StartMin,DC1_to_LN31_Messages[14]) ,MID(LN31_Weekly_Schedule.Monday._3rd_Shift_End,2,1,CurrentSchedule.s3EndHour) STOD(CurrentSchedule.s3EndHour,DC1_to_LN31_Messages[15]) MID(LN31_Weekly_Schedule.Monday._3rd_Shift_End,2,4,CurrentSchedule.s3EndMin) STOD(CurrentSchedule.s3EndMin,DC1_to_LN31_Messages[16]) ];
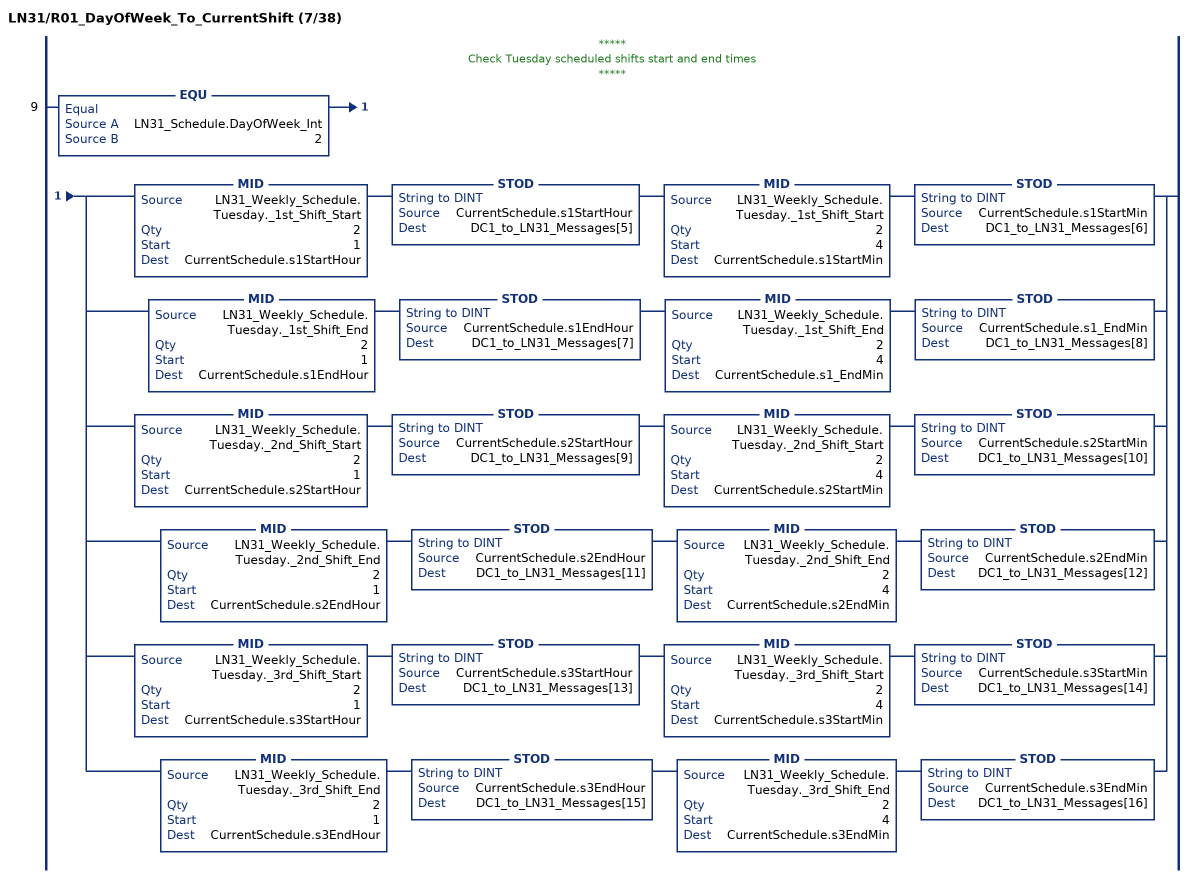
   // *****
   // Check Tuesday scheduled shifts start and end times
   // *****
   9: EQU(LN31_Schedule.DayOfWeek_Int,2)[MID(LN31_Weekly_Schedule.Tuesday._1st_Shift_Start,2,1,CurrentSchedule.s1StartHour) STOD(CurrentSchedule.s1StartHour,DC1_to_LN31_Messages[5]) MID(LN31_Weekly_Schedule.Tuesday._1st_Shift_Start,2,4,CurrentSchedule.s1StartMin) STOD(CurrentSchedule.s1StartMin,DC1_to_LN31_Messages[6]) ,MID(LN31_Weekly_Schedule.Tuesday._1st_Shift_End,2,1,CurrentSchedule.s1EndHour) STOD(CurrentSchedule.s1EndHour,DC1_to_LN31_Messages[7]) MID(LN31_Weekly_Schedule.Tuesday._1st_Shift_End,2,4,CurrentSchedule.s1_EndMin) STOD(CurrentSchedule.s1_EndMin,DC1_to_LN31_Messages[8]) ,MID(LN31_Weekly_Schedule.Tuesday._2nd_Shift_Start,2,1,CurrentSchedule.s2StartHour) STOD(CurrentSchedule.s2StartHour,DC1_to_LN31_Messages[9]) MID(LN31_Weekly_Schedule.Tuesday._2nd_Shift_Start,2,4,CurrentSchedule.s2StartMin) STOD(CurrentSchedule.s2StartMin,DC1_to_LN31_Messages[10]) ,MID(LN31_Weekly_Schedule.Tuesday._2nd_Shift_End,2,1,CurrentSchedule.s2EndHour) STOD(CurrentSchedule.s2EndHour,DC1_to_LN31_Messages[11]) MID(LN31_Weekly_Schedule.Tuesday._2nd_Shift_End,2,4,CurrentSchedule.s2EndMin) STOD(CurrentSchedule.s2EndMin,DC1_to_LN31_Messages[12]) ,MID(LN31_Weekly_Schedule.Tuesday._3rd_Shift_Start,2,1,CurrentSchedule.s3StartHour) STOD(CurrentSchedule.s3StartHour,DC1_to_LN31_Messages[13]) MID(LN31_Weekly_Schedule.Tuesday._3rd_Shift_Start,2,4,CurrentSchedule.s3StartMin) STOD(CurrentSchedule.s3StartMin,DC1_to_LN31_Messages[14]) ,MID(LN31_Weekly_Schedule.Tuesday._3rd_Shift_End,2,1,CurrentSchedule.s3EndHour) STOD(CurrentSchedule.s3EndHour,DC1_to_LN31_Messages[15]) MID(LN31_Weekly_Schedule.Tuesday._3rd_Shift_End,2,4,CurrentSchedule.s3EndMin) STOD(CurrentSchedule.s3EndMin,DC1_to_LN31_Messages[16]) ];
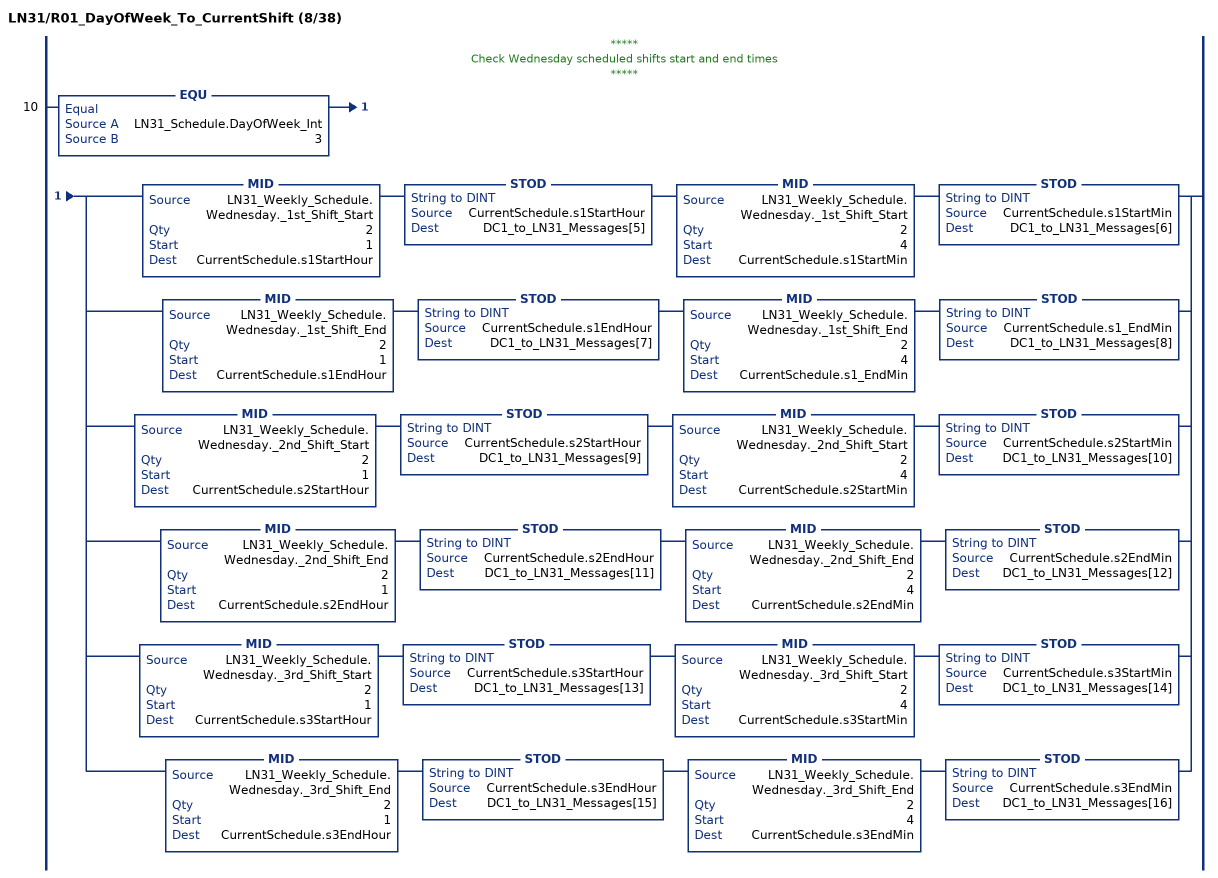
   // *****
   // Check Wednesday scheduled shifts start and end times
   // *****
   10: EQU(LN31_Schedule.DayOfWeek_Int,3)[MID(LN31_Weekly_Schedule.Wednesday._1st_Shift_Start,2,1,CurrentSchedule.s1StartHour) STOD(CurrentSchedule.s1StartHour,DC1_to_LN31_Messages[5]) MID(LN31_Weekly_Schedule.Wednesday._1st_Shift_Start,2,4,CurrentSchedule.s1StartMin) STOD(CurrentSchedule.s1StartMin,DC1_to_LN31_Messages[6]) ,MID(LN31_Weekly_Schedule.Wednesday._1st_Shift_End,2,1,CurrentSchedule.s1EndHour) STOD(CurrentSchedule.s1EndHour,DC1_to_LN31_Messages[7]) MID(LN31_Weekly_Schedule.Wednesday._1st_Shift_End,2,4,CurrentSchedule.s1_EndMin) STOD(CurrentSchedule.s1_EndMin,DC1_to_LN31_Messages[8]) ,MID(LN31_Weekly_Schedule.Wednesday._2nd_Shift_Start,2,1,CurrentSchedule.s2StartHour) STOD(CurrentSchedule.s2StartHour,DC1_to_LN31_Messages[9]) MID(LN31_Weekly_Schedule.Wednesday._2nd_Shift_Start,2,4,CurrentSchedule.s2StartMin) STOD(CurrentSchedule.s2StartMin,DC1_to_LN31_Messages[10]) ,MID(LN31_Weekly_Schedule.Wednesday._2nd_Shift_End,2,1,CurrentSchedule.s2EndHour) STOD(CurrentSchedule.s2EndHour,DC1_to_LN31_Messages[11]) MID(LN31_Weekly_Schedule.Wednesday._2nd_Shift_End,2,4,CurrentSchedule.s2EndMin) STOD(CurrentSchedule.s2EndMin,DC1_to_LN31_Messages[12]) ,MID(LN31_Weekly_Schedule.Wednesday._3rd_Shift_Start,2,1,CurrentSchedule.s3StartHour) STOD(CurrentSchedule.s3StartHour,DC1_to_LN31_Messages[13]) MID(LN31_Weekly_Schedule.Wednesday._3rd_Shift_Start,2,4,CurrentSchedule.s3StartMin) STOD(CurrentSchedule.s3StartMin,DC1_to_LN31_Messages[14]) ,MID(LN31_Weekly_Schedule.Wednesday._3rd_Shift_End,2,1,CurrentSchedule.s3EndHour) STOD(CurrentSchedule.s3EndHour,DC1_to_LN31_Messages[15]) MID(LN31_Weekly_Schedule.Wednesday._3rd_Shift_End,2,4,CurrentSchedule.s3EndMin) STOD(CurrentSchedule.s3EndMin,DC1_to_LN31_Messages[16]) ];
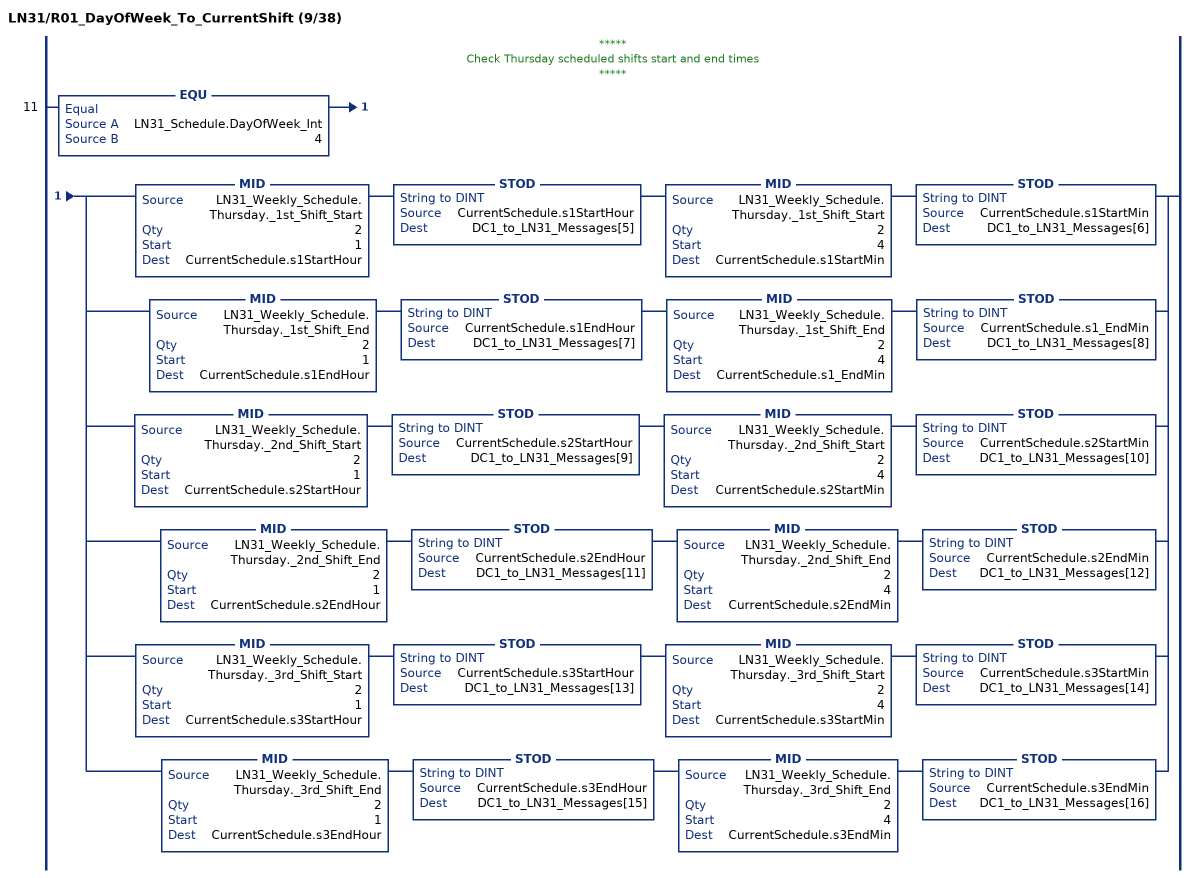
   // *****
   // Check Thursday scheduled shifts start and end times
   // *****
   11: EQU(LN31_Schedule.DayOfWeek_Int,4)[MID(LN31_Weekly_Schedule.Thursday._1st_Shift_Start,2,1,CurrentSchedule.s1StartHour) STOD(CurrentSchedule.s1StartHour,DC1_to_LN31_Messages[5]) MID(LN31_Weekly_Schedule.Thursday._1st_Shift_Start,2,4,CurrentSchedule.s1StartMin) STOD(CurrentSchedule.s1StartMin,DC1_to_LN31_Messages[6]) ,MID(LN31_Weekly_Schedule.Thursday._1st_Shift_End,2,1,CurrentSchedule.s1EndHour) STOD(CurrentSchedule.s1EndHour,DC1_to_LN31_Messages[7]) MID(LN31_Weekly_Schedule.Thursday._1st_Shift_End,2,4,CurrentSchedule.s1_EndMin) STOD(CurrentSchedule.s1_EndMin,DC1_to_LN31_Messages[8]) ,MID(LN31_Weekly_Schedule.Thursday._2nd_Shift_Start,2,1,CurrentSchedule.s2StartHour) STOD(CurrentSchedule.s2StartHour,DC1_to_LN31_Messages[9]) MID(LN31_Weekly_Schedule.Thursday._2nd_Shift_Start,2,4,CurrentSchedule.s2StartMin) STOD(CurrentSchedule.s2StartMin,DC1_to_LN31_Messages[10]) ,MID(LN31_Weekly_Schedule.Thursday._2nd_Shift_End,2,1,CurrentSchedule.s2EndHour) STOD(CurrentSchedule.s2EndHour,DC1_to_LN31_Messages[11]) MID(LN31_Weekly_Schedule.Thursday._2nd_Shift_End,2,4,CurrentSchedule.s2EndMin) STOD(CurrentSchedule.s2EndMin,DC1_to_LN31_Messages[12]) ,MID(LN31_Weekly_Schedule.Thursday._3rd_Shift_Start,2,1,CurrentSchedule.s3StartHour) STOD(CurrentSchedule.s3StartHour,DC1_to_LN31_Messages[13]) MID(LN31_Weekly_Schedule.Thursday._3rd_Shift_Start,2,4,CurrentSchedule.s3StartMin) STOD(CurrentSchedule.s3StartMin,DC1_to_LN31_Messages[14]) ,MID(LN31_Weekly_Schedule.Thursday._3rd_Shift_End,2,1,CurrentSchedule.s3EndHour) STOD(CurrentSchedule.s3EndHour,DC1_to_LN31_Messages[15]) MID(LN31_Weekly_Schedule.Thursday._3rd_Shift_End,2,4,CurrentSchedule.s3EndMin) STOD(CurrentSchedule.s3EndMin,DC1_to_LN31_Messages[16]) ];
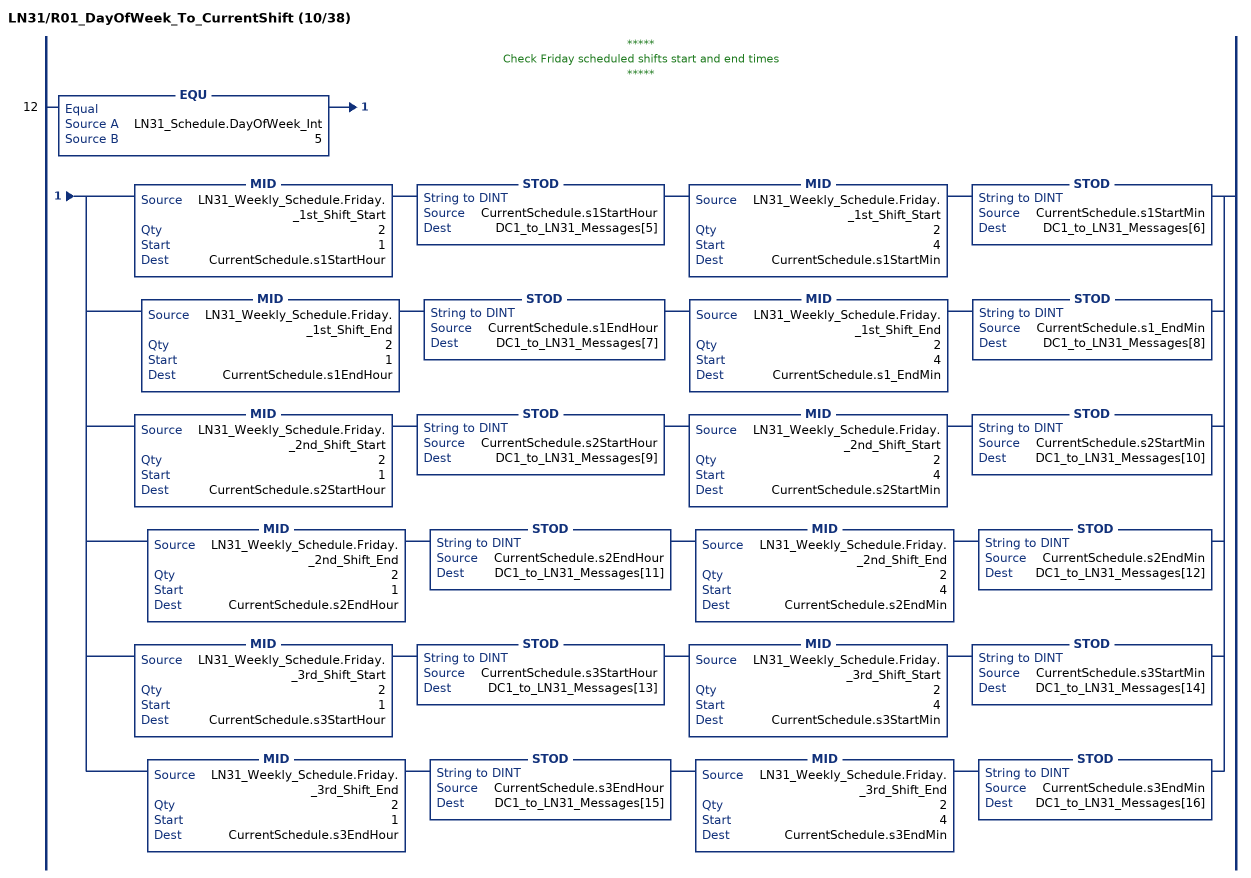
   // *****
   // Check Friday scheduled shifts start and end times
   // *****
   12: EQU(LN31_Schedule.DayOfWeek_Int,5)[MID(LN31_Weekly_Schedule.Friday._1st_Shift_Start,2,1,CurrentSchedule.s1StartHour) STOD(CurrentSchedule.s1StartHour,DC1_to_LN31_Messages[5]) MID(LN31_Weekly_Schedule.Friday._1st_Shift_Start,2,4,CurrentSchedule.s1StartMin) STOD(CurrentSchedule.s1StartMin,DC1_to_LN31_Messages[6]) ,MID(LN31_Weekly_Schedule.Friday._1st_Shift_End,2,1,CurrentSchedule.s1EndHour) STOD(CurrentSchedule.s1EndHour,DC1_to_LN31_Messages[7]) MID(LN31_Weekly_Schedule.Friday._1st_Shift_End,2,4,CurrentSchedule.s1_EndMin) STOD(CurrentSchedule.s1_EndMin,DC1_to_LN31_Messages[8]) ,MID(LN31_Weekly_Schedule.Friday._2nd_Shift_Start,2,1,CurrentSchedule.s2StartHour) STOD(CurrentSchedule.s2StartHour,DC1_to_LN31_Messages[9]) MID(LN31_Weekly_Schedule.Friday._2nd_Shift_Start,2,4,CurrentSchedule.s2StartMin) STOD(CurrentSchedule.s2StartMin,DC1_to_LN31_Messages[10]) ,MID(LN31_Weekly_Schedule.Friday._2nd_Shift_End,2,1,CurrentSchedule.s2EndHour) STOD(CurrentSchedule.s2EndHour,DC1_to_LN31_Messages[11]) MID(LN31_Weekly_Schedule.Friday._2nd_Shift_End,2,4,CurrentSchedule.s2EndMin) STOD(CurrentSchedule.s2EndMin,DC1_to_LN31_Messages[12]) ,MID(LN31_Weekly_Schedule.Friday._3rd_Shift_Start,2,1,CurrentSchedule.s3StartHour) STOD(CurrentSchedule.s3StartHour,DC1_to_LN31_Messages[13]) MID(LN31_Weekly_Schedule.Friday._3rd_Shift_Start,2,4,CurrentSchedule.s3StartMin) STOD(CurrentSchedule.s3StartMin,DC1_to_LN31_Messages[14]) ,MID(LN31_Weekly_Schedule.Friday._3rd_Shift_End,2,1,CurrentSchedule.s3EndHour) STOD(CurrentSchedule.s3EndHour,DC1_to_LN31_Messages[15]) MID(LN31_Weekly_Schedule.Friday._3rd_Shift_End,2,4,CurrentSchedule.s3EndMin) STOD(CurrentSchedule.s3EndMin,DC1_to_LN31_Messages[16]) ];
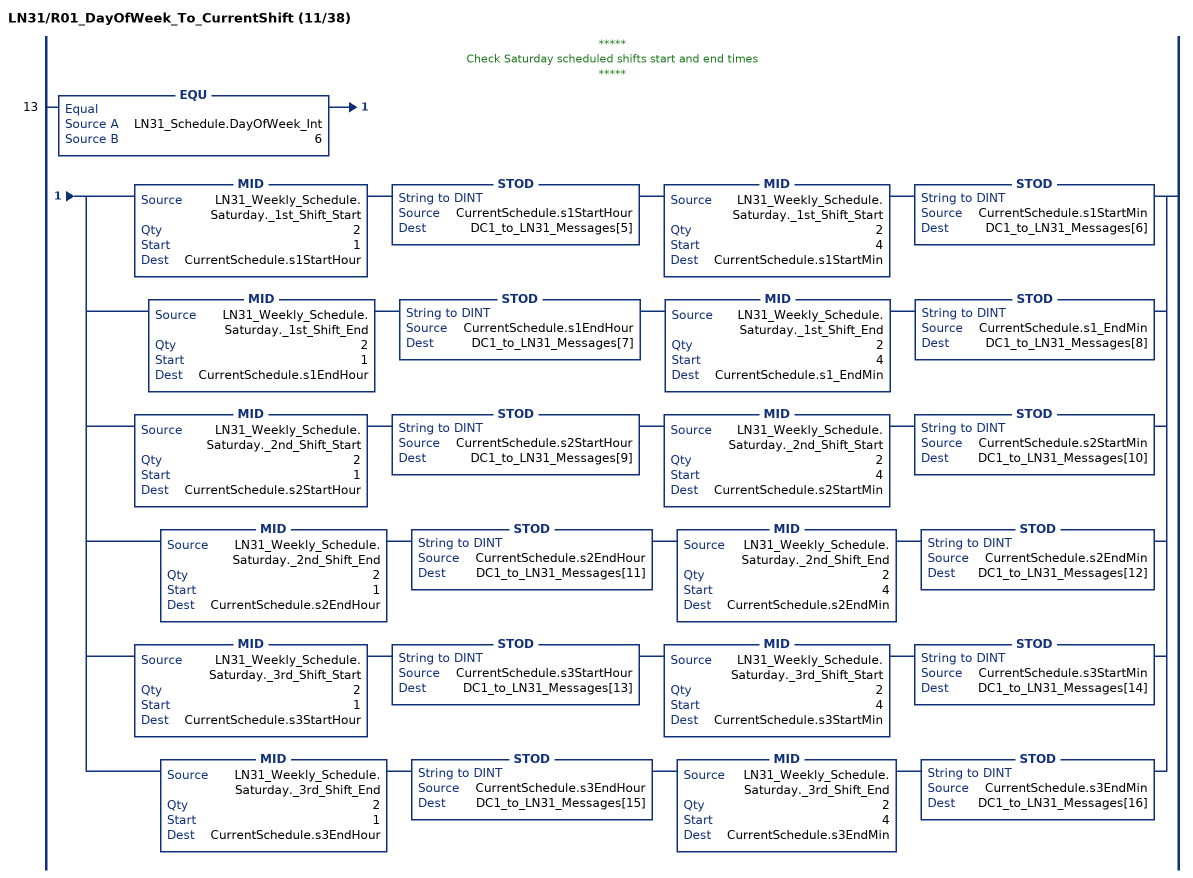
   // *****
   // Check Saturday scheduled shifts start and end times
   // *****
   13: EQU(LN31_Schedule.DayOfWeek_Int,6)[MID(LN31_Weekly_Schedule.Saturday._1st_Shift_Start,2,1,CurrentSchedule.s1StartHour) STOD(CurrentSchedule.s1StartHour,DC1_to_LN31_Messages[5]) MID(LN31_Weekly_Schedule.Saturday._1st_Shift_Start,2,4,CurrentSchedule.s1StartMin) STOD(CurrentSchedule.s1StartMin,DC1_to_LN31_Messages[6]) ,MID(LN31_Weekly_Schedule.Saturday._1st_Shift_End,2,1,CurrentSchedule.s1EndHour) STOD(CurrentSchedule.s1EndHour,DC1_to_LN31_Messages[7]) MID(LN31_Weekly_Schedule.Saturday._1st_Shift_End,2,4,CurrentSchedule.s1_EndMin) STOD(CurrentSchedule.s1_EndMin,DC1_to_LN31_Messages[8]) ,MID(LN31_Weekly_Schedule.Saturday._2nd_Shift_Start,2,1,CurrentSchedule.s2StartHour) STOD(CurrentSchedule.s2StartHour,DC1_to_LN31_Messages[9]) MID(LN31_Weekly_Schedule.Saturday._2nd_Shift_Start,2,4,CurrentSchedule.s2StartMin) STOD(CurrentSchedule.s2StartMin,DC1_to_LN31_Messages[10]) ,MID(LN31_Weekly_Schedule.Saturday._2nd_Shift_End,2,1,CurrentSchedule.s2EndHour) STOD(CurrentSchedule.s2EndHour,DC1_to_LN31_Messages[11]) MID(LN31_Weekly_Schedule.Saturday._2nd_Shift_End,2,4,CurrentSchedule.s2EndMin) STOD(CurrentSchedule.s2EndMin,DC1_to_LN31_Messages[12]) ,MID(LN31_Weekly_Schedule.Saturday._3rd_Shift_Start,2,1,CurrentSchedule.s3StartHour) STOD(CurrentSchedule.s3StartHour,DC1_to_LN31_Messages[13]) MID(LN31_Weekly_Schedule.Saturday._3rd_Shift_Start,2,4,CurrentSchedule.s3StartMin) STOD(CurrentSchedule.s3StartMin,DC1_to_LN31_Messages[14]) ,MID(LN31_Weekly_Schedule.Saturday._3rd_Shift_End,2,1,CurrentSchedule.s3EndHour) STOD(CurrentSchedule.s3EndHour,DC1_to_LN31_Messages[15]) MID(LN31_Weekly_Schedule.Saturday._3rd_Shift_End,2,4,CurrentSchedule.s3EndMin) STOD(CurrentSchedule.s3EndMin,DC1_to_LN31_Messages[16]) ];
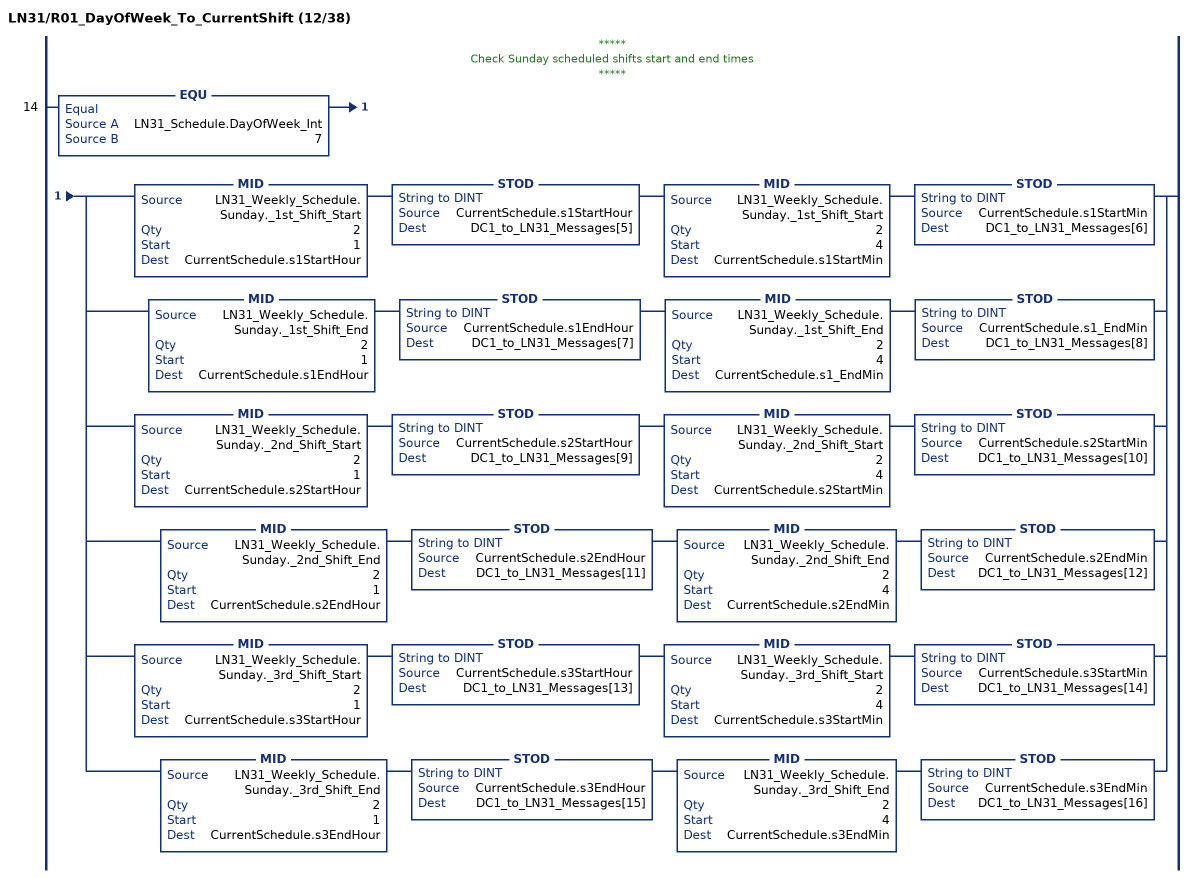
   // *****
   // Check Sunday scheduled shifts start and end times
   // *****
   14: EQU(LN31_Schedule.DayOfWeek_Int,7)[MID(LN31_Weekly_Schedule.Sunday._1st_Shift_Start,2,1,CurrentSchedule.s1StartHour) STOD(CurrentSchedule.s1StartHour,DC1_to_LN31_Messages[5]) MID(LN31_Weekly_Schedule.Sunday._1st_Shift_Start,2,4,CurrentSchedule.s1StartMin) STOD(CurrentSchedule.s1StartMin,DC1_to_LN31_Messages[6]) ,MID(LN31_Weekly_Schedule.Sunday._1st_Shift_End,2,1,CurrentSchedule.s1EndHour) STOD(CurrentSchedule.s1EndHour,DC1_to_LN31_Messages[7]) MID(LN31_Weekly_Schedule.Sunday._1st_Shift_End,2,4,CurrentSchedule.s1_EndMin) STOD(CurrentSchedule.s1_EndMin,DC1_to_LN31_Messages[8]) ,MID(LN31_Weekly_Schedule.Sunday._2nd_Shift_Start,2,1,CurrentSchedule.s2StartHour) STOD(CurrentSchedule.s2StartHour,DC1_to_LN31_Messages[9]) MID(LN31_Weekly_Schedule.Sunday._2nd_Shift_Start,2,4,CurrentSchedule.s2StartMin) STOD(CurrentSchedule.s2StartMin,DC1_to_LN31_Messages[10]) ,MID(LN31_Weekly_Schedule.Sunday._2nd_Shift_End,2,1,CurrentSchedule.s2EndHour) STOD(CurrentSchedule.s2EndHour,DC1_to_LN31_Messages[11]) MID(LN31_Weekly_Schedule.Sunday._2nd_Shift_End,2,4,CurrentSchedule.s2EndMin) STOD(CurrentSchedule.s2EndMin,DC1_to_LN31_Messages[12]) ,MID(LN31_Weekly_Schedule.Sunday._3rd_Shift_Start,2,1,CurrentSchedule.s3StartHour) STOD(CurrentSchedule.s3StartHour,DC1_to_LN31_Messages[13]) MID(LN31_Weekly_Schedule.Sunday._3rd_Shift_Start,2,4,CurrentSchedule.s3StartMin) STOD(CurrentSchedule.s3StartMin,DC1_to_LN31_Messages[14]) ,MID(LN31_Weekly_Schedule.Sunday._3rd_Shift_End,2,1,CurrentSchedule.s3EndHour) STOD(CurrentSchedule.s3EndHour,DC1_to_LN31_Messages[15]) MID(LN31_Weekly_Schedule.Sunday._3rd_Shift_End,2,4,CurrentSchedule.s3EndMin) STOD(CurrentSchedule.s3EndMin,DC1_to_LN31_Messages[16]) ];
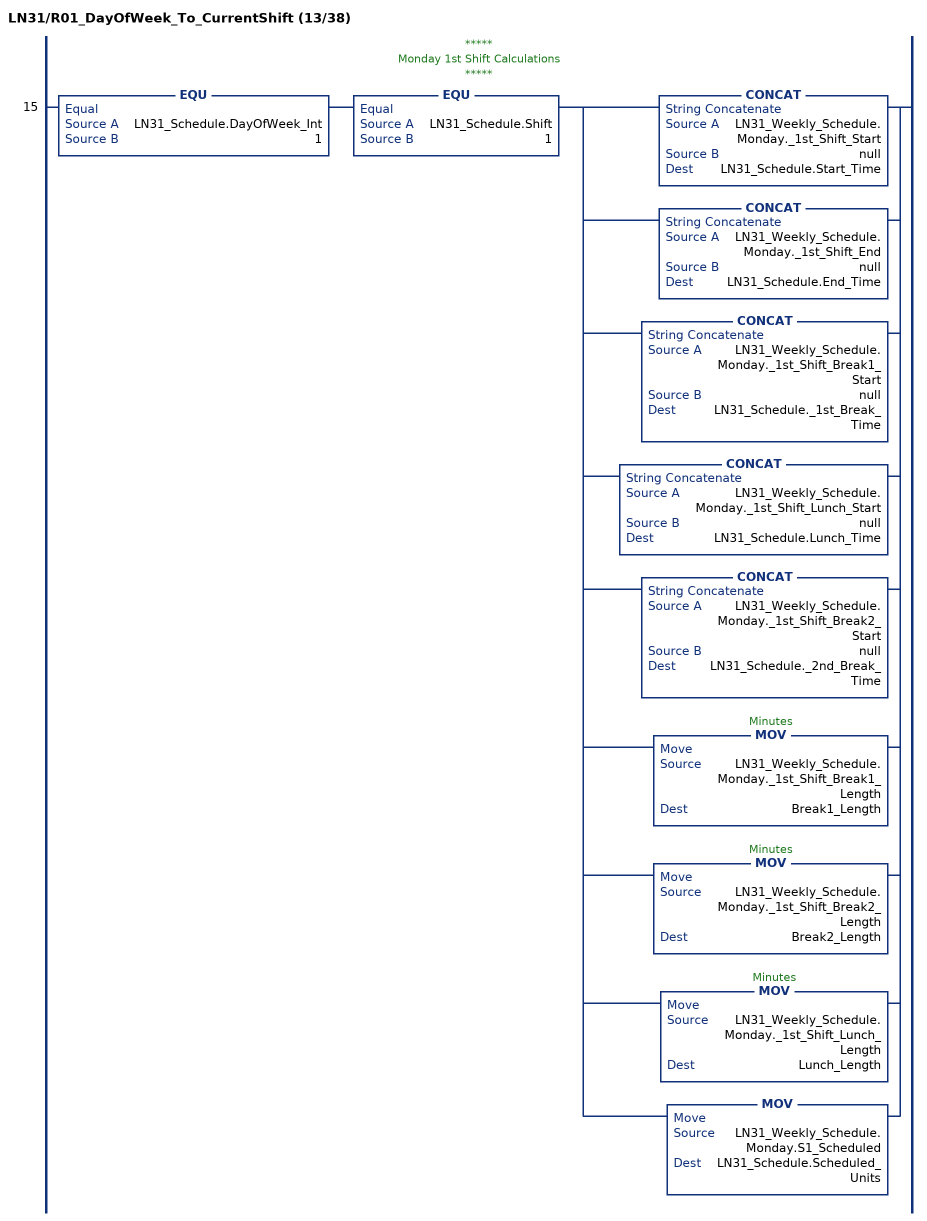
   // *****
   // Monday 1st Shift Calculations
   // *****
   15: EQU(LN31_Schedule.DayOfWeek_Int,1)EQU(LN31_Schedule.Shift,1)[CONCAT(LN31_Weekly_Schedule.Monday._1st_Shift_Start,null,LN31_Schedule.Start_Time) ,CONCAT(LN31_Weekly_Schedule.Monday._1st_Shift_End,null,LN31_Schedule.End_Time) ,CONCAT(LN31_Weekly_Schedule.Monday._1st_Shift_Break1_Start,null,LN31_Schedule._1st_Break_Time) ,CONCAT(LN31_Weekly_Schedule.Monday._1st_Shift_Lunch_Start,null,LN31_Schedule.Lunch_Time) ,CONCAT(LN31_Weekly_Schedule.Monday._1st_Shift_Break2_Start,null,LN31_Schedule._2nd_Break_Time) ,MOV(LN31_Weekly_Schedule.Monday._1st_Shift_Break1_Length,Break1_Length) ,MOV(LN31_Weekly_Schedule.Monday._1st_Shift_Break2_Length,Break2_Length) ,MOV(LN31_Weekly_Schedule.Monday._1st_Shift_Lunch_Length,Lunch_Length) ,MOV(LN31_Weekly_Schedule.Monday.S1_Scheduled,LN31_Schedule.Scheduled_Units) ];
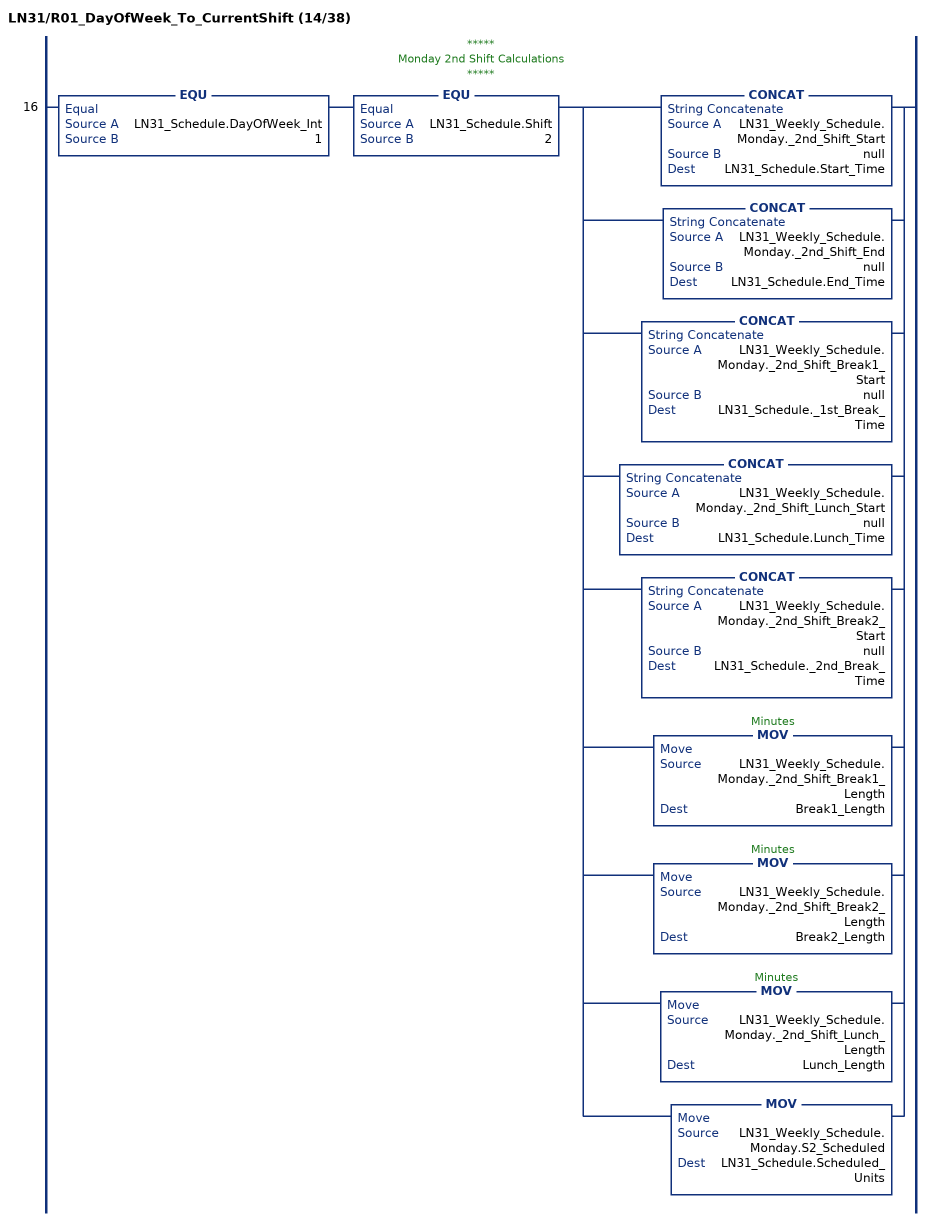
   // *****
   // Monday 2nd Shift Calculations
   // *****
   16: EQU(LN31_Schedule.DayOfWeek_Int,1)EQU(LN31_Schedule.Shift,2)[CONCAT(LN31_Weekly_Schedule.Monday._2nd_Shift_Start,null,LN31_Schedule.Start_Time) ,CONCAT(LN31_Weekly_Schedule.Monday._2nd_Shift_End,null,LN31_Schedule.End_Time) ,CONCAT(LN31_Weekly_Schedule.Monday._2nd_Shift_Break1_Start,null,LN31_Schedule._1st_Break_Time) ,CONCAT(LN31_Weekly_Schedule.Monday._2nd_Shift_Lunch_Start,null,LN31_Schedule.Lunch_Time) ,CONCAT(LN31_Weekly_Schedule.Monday._2nd_Shift_Break2_Start,null,LN31_Schedule._2nd_Break_Time) ,MOV(LN31_Weekly_Schedule.Monday._2nd_Shift_Break1_Length,Break1_Length) ,MOV(LN31_Weekly_Schedule.Monday._2nd_Shift_Break2_Length,Break2_Length) ,MOV(LN31_Weekly_Schedule.Monday._2nd_Shift_Lunch_Length,Lunch_Length) ,MOV(LN31_Weekly_Schedule.Monday.S2_Scheduled,LN31_Schedule.Scheduled_Units) ];
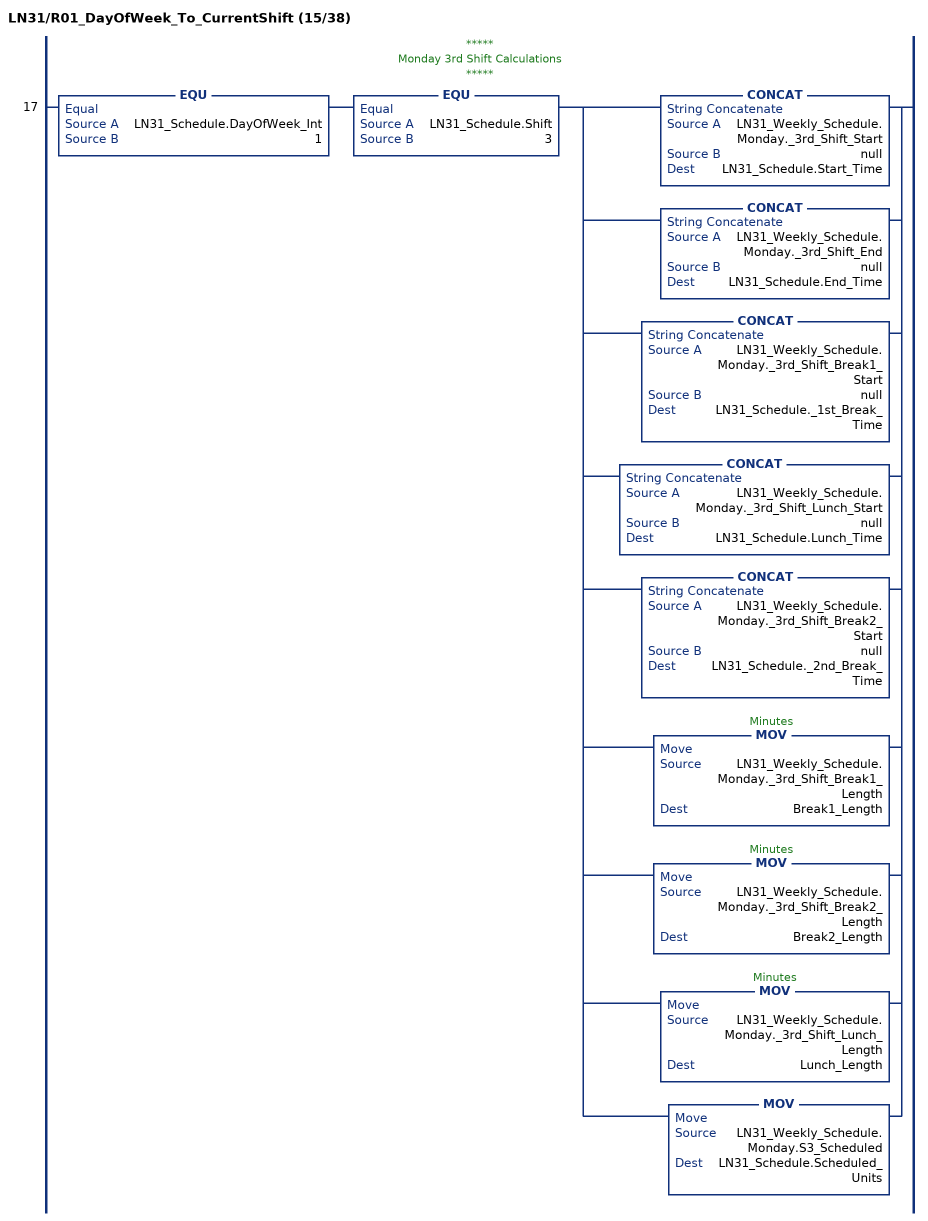
   // *****
   // Monday 3rd Shift Calculations
   // *****
   17: EQU(LN31_Schedule.DayOfWeek_Int,1)EQU(LN31_Schedule.Shift,3)[CONCAT(LN31_Weekly_Schedule.Monday._3rd_Shift_Start,null,LN31_Schedule.Start_Time) ,CONCAT(LN31_Weekly_Schedule.Monday._3rd_Shift_End,null,LN31_Schedule.End_Time) ,CONCAT(LN31_Weekly_Schedule.Monday._3rd_Shift_Break1_Start,null,LN31_Schedule._1st_Break_Time) ,CONCAT(LN31_Weekly_Schedule.Monday._3rd_Shift_Lunch_Start,null,LN31_Schedule.Lunch_Time) ,CONCAT(LN31_Weekly_Schedule.Monday._3rd_Shift_Break2_Start,null,LN31_Schedule._2nd_Break_Time) ,MOV(LN31_Weekly_Schedule.Monday._3rd_Shift_Break1_Length,Break1_Length) ,MOV(LN31_Weekly_Schedule.Monday._3rd_Shift_Break2_Length,Break2_Length) ,MOV(LN31_Weekly_Schedule.Monday._3rd_Shift_Lunch_Length,Lunch_Length) ,MOV(LN31_Weekly_Schedule.Monday.S3_Scheduled,LN31_Schedule.Scheduled_Units) ];
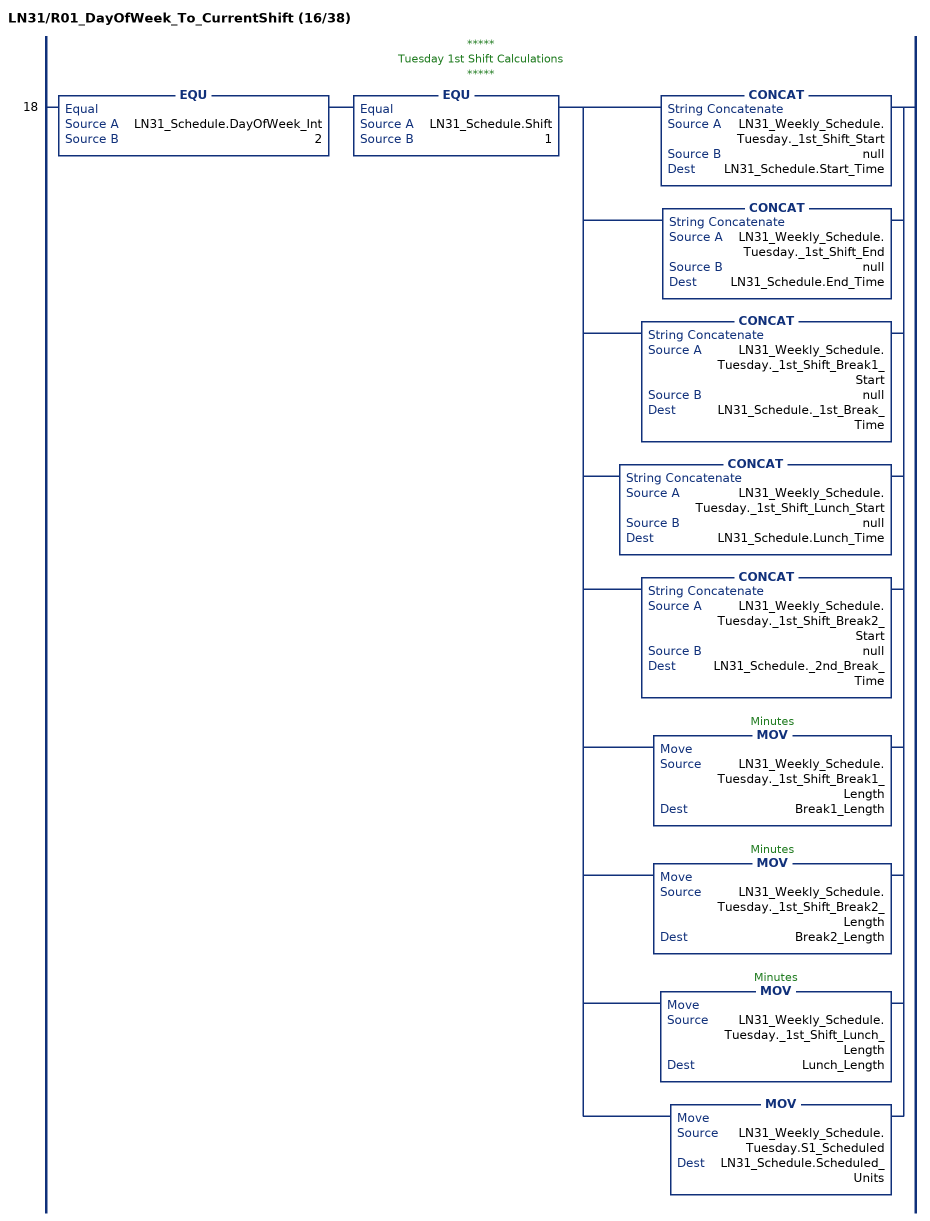
   // *****
   // Tuesday 1st Shift Calculations
   // *****
   18: EQU(LN31_Schedule.DayOfWeek_Int,2)EQU(LN31_Schedule.Shift,1)[CONCAT(LN31_Weekly_Schedule.Tuesday._1st_Shift_Start,null,LN31_Schedule.Start_Time) ,CONCAT(LN31_Weekly_Schedule.Tuesday._1st_Shift_End,null,LN31_Schedule.End_Time) ,CONCAT(LN31_Weekly_Schedule.Tuesday._1st_Shift_Break1_Start,null,LN31_Schedule._1st_Break_Time) ,CONCAT(LN31_Weekly_Schedule.Tuesday._1st_Shift_Lunch_Start,null,LN31_Schedule.Lunch_Time) ,CONCAT(LN31_Weekly_Schedule.Tuesday._1st_Shift_Break2_Start,null,LN31_Schedule._2nd_Break_Time) ,MOV(LN31_Weekly_Schedule.Tuesday._1st_Shift_Break1_Length,Break1_Length) ,MOV(LN31_Weekly_Schedule.Tuesday._1st_Shift_Break2_Length,Break2_Length) ,MOV(LN31_Weekly_Schedule.Tuesday._1st_Shift_Lunch_Length,Lunch_Length) ,MOV(LN31_Weekly_Schedule.Tuesday.S1_Scheduled,LN31_Schedule.Scheduled_Units) ];
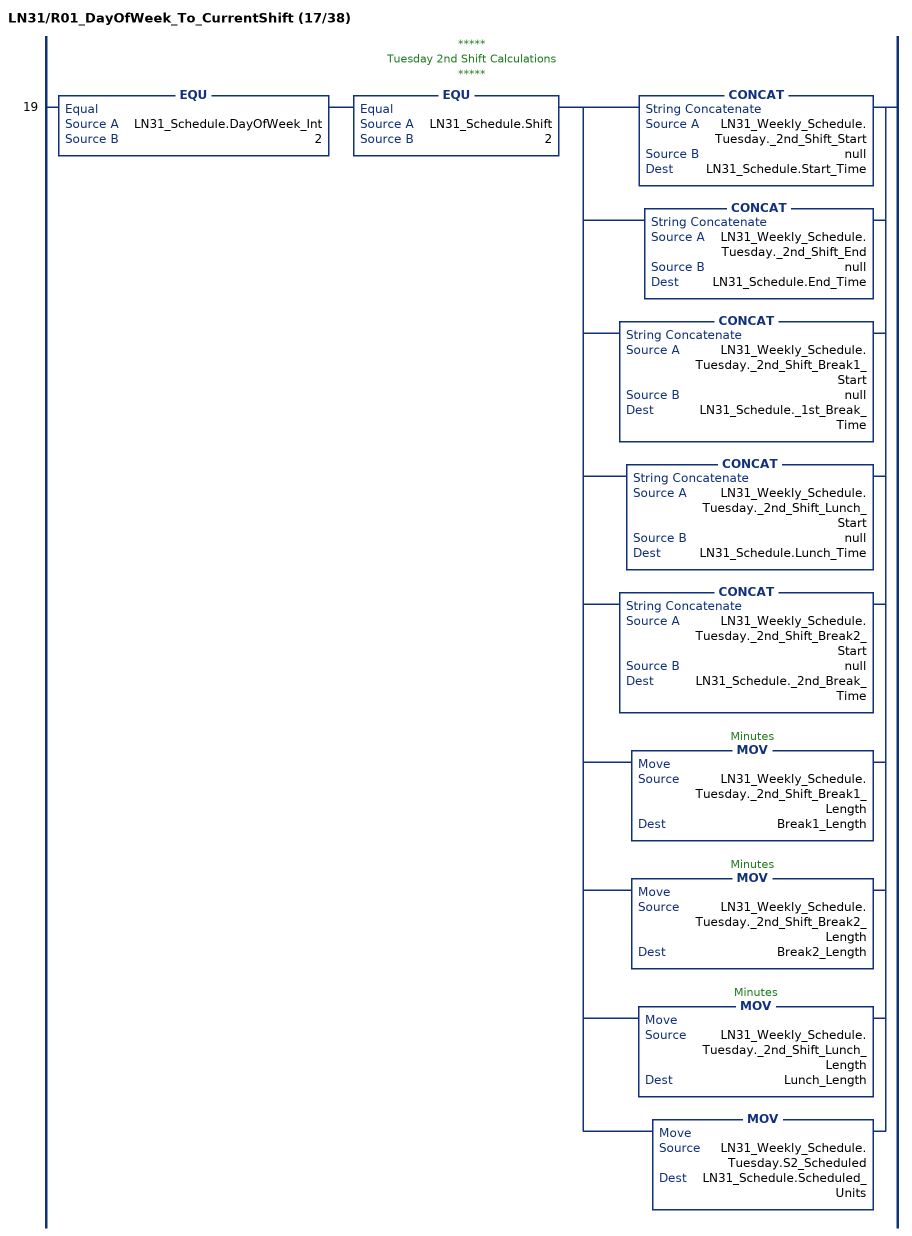
   // *****
   // Tuesday 2nd Shift Calculations
   // *****
   19: EQU(LN31_Schedule.DayOfWeek_Int,2)EQU(LN31_Schedule.Shift,2)[CONCAT(LN31_Weekly_Schedule.Tuesday._2nd_Shift_Start,null,LN31_Schedule.Start_Time) ,CONCAT(LN31_Weekly_Schedule.Tuesday._2nd_Shift_End,null,LN31_Schedule.End_Time) ,CONCAT(LN31_Weekly_Schedule.Tuesday._2nd_Shift_Break1_Start,null,LN31_Schedule._1st_Break_Time) ,CONCAT(LN31_Weekly_Schedule.Tuesday._2nd_Shift_Lunch_Start,null,LN31_Schedule.Lunch_Time) ,CONCAT(LN31_Weekly_Schedule.Tuesday._2nd_Shift_Break2_Start,null,LN31_Schedule._2nd_Break_Time) ,MOV(LN31_Weekly_Schedule.Tuesday._2nd_Shift_Break1_Length,Break1_Length) ,MOV(LN31_Weekly_Schedule.Tuesday._2nd_Shift_Break2_Length,Break2_Length) ,MOV(LN31_Weekly_Schedule.Tuesday._2nd_Shift_Lunch_Length,Lunch_Length) ,MOV(LN31_Weekly_Schedule.Tuesday.S2_Scheduled,LN31_Schedule.Scheduled_Units) ];
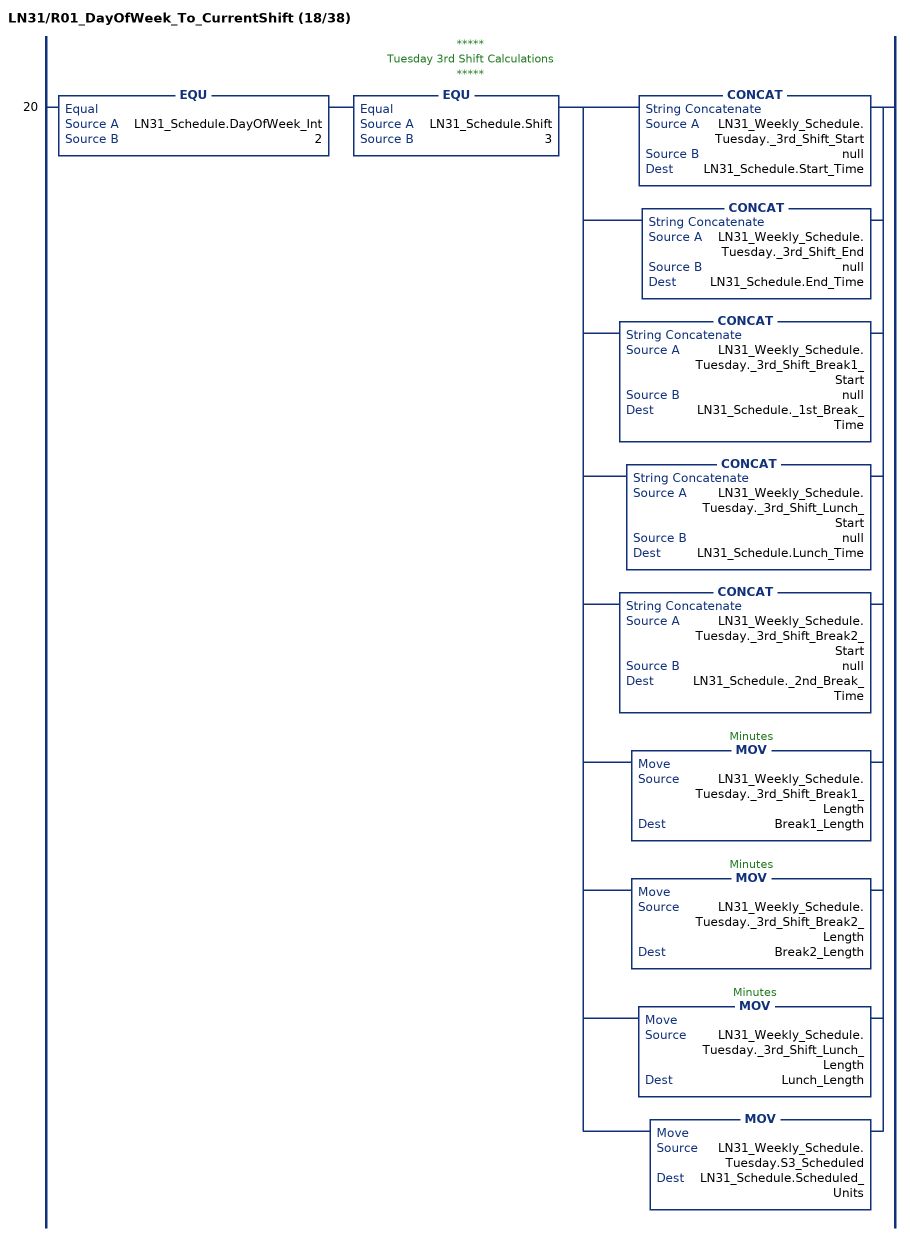
   // *****
   // Tuesday 3rd Shift Calculations
   // *****
   20: EQU(LN31_Schedule.DayOfWeek_Int,2)EQU(LN31_Schedule.Shift,3)[CONCAT(LN31_Weekly_Schedule.Tuesday._3rd_Shift_Start,null,LN31_Schedule.Start_Time) ,CONCAT(LN31_Weekly_Schedule.Tuesday._3rd_Shift_End,null,LN31_Schedule.End_Time) ,CONCAT(LN31_Weekly_Schedule.Tuesday._3rd_Shift_Break1_Start,null,LN31_Schedule._1st_Break_Time) ,CONCAT(LN31_Weekly_Schedule.Tuesday._3rd_Shift_Lunch_Start,null,LN31_Schedule.Lunch_Time) ,CONCAT(LN31_Weekly_Schedule.Tuesday._3rd_Shift_Break2_Start,null,LN31_Schedule._2nd_Break_Time) ,MOV(LN31_Weekly_Schedule.Tuesday._3rd_Shift_Break1_Length,Break1_Length) ,MOV(LN31_Weekly_Schedule.Tuesday._3rd_Shift_Break2_Length,Break2_Length) ,MOV(LN31_Weekly_Schedule.Tuesday._3rd_Shift_Lunch_Length,Lunch_Length) ,MOV(LN31_Weekly_Schedule.Tuesday.S3_Scheduled,LN31_Schedule.Scheduled_Units) ];
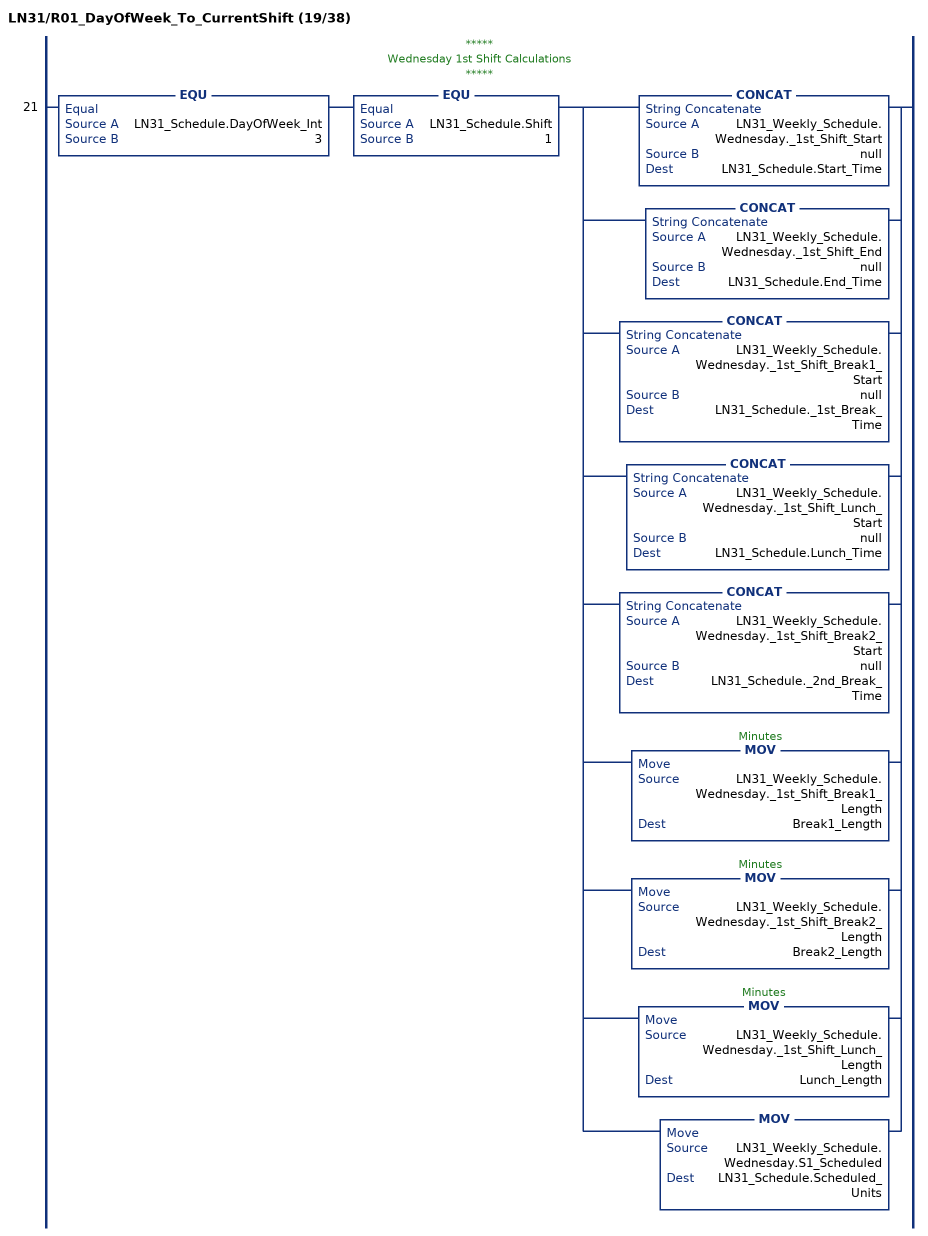
   // *****
   // Wednesday 1st Shift Calculations
   // *****
   21: EQU(LN31_Schedule.DayOfWeek_Int,3)EQU(LN31_Schedule.Shift,1)[CONCAT(LN31_Weekly_Schedule.Wednesday._1st_Shift_Start,null,LN31_Schedule.Start_Time) ,CONCAT(LN31_Weekly_Schedule.Wednesday._1st_Shift_End,null,LN31_Schedule.End_Time) ,CONCAT(LN31_Weekly_Schedule.Wednesday._1st_Shift_Break1_Start,null,LN31_Schedule._1st_Break_Time) ,CONCAT(LN31_Weekly_Schedule.Wednesday._1st_Shift_Lunch_Start,null,LN31_Schedule.Lunch_Time) ,CONCAT(LN31_Weekly_Schedule.Wednesday._1st_Shift_Break2_Start,null,LN31_Schedule._2nd_Break_Time) ,MOV(LN31_Weekly_Schedule.Wednesday._1st_Shift_Break1_Length,Break1_Length) ,MOV(LN31_Weekly_Schedule.Wednesday._1st_Shift_Break2_Length,Break2_Length) ,MOV(LN31_Weekly_Schedule.Wednesday._1st_Shift_Lunch_Length,Lunch_Length) ,MOV(LN31_Weekly_Schedule.Wednesday.S1_Scheduled,LN31_Schedule.Scheduled_Units) ];
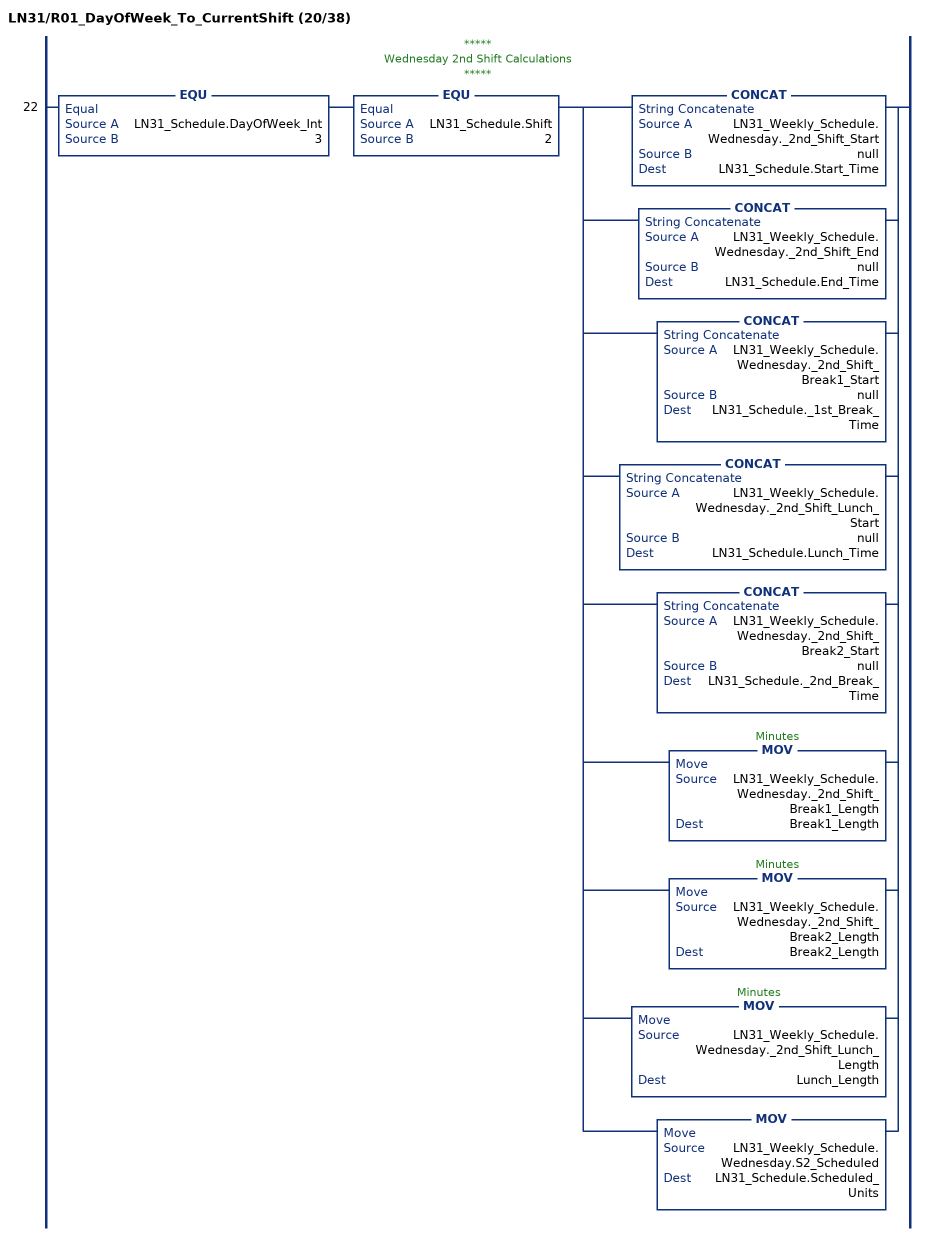
   // *****
   // Wednesday 2nd Shift Calculations
   // *****
   22: EQU(LN31_Schedule.DayOfWeek_Int,3)EQU(LN31_Schedule.Shift,2)[CONCAT(LN31_Weekly_Schedule.Wednesday._2nd_Shift_Start,null,LN31_Schedule.Start_Time) ,CONCAT(LN31_Weekly_Schedule.Wednesday._2nd_Shift_End,null,LN31_Schedule.End_Time) ,CONCAT(LN31_Weekly_Schedule.Wednesday._2nd_Shift_Break1_Start,null,LN31_Schedule._1st_Break_Time) ,CONCAT(LN31_Weekly_Schedule.Wednesday._2nd_Shift_Lunch_Start,null,LN31_Schedule.Lunch_Time) ,CONCAT(LN31_Weekly_Schedule.Wednesday._2nd_Shift_Break2_Start,null,LN31_Schedule._2nd_Break_Time) ,MOV(LN31_Weekly_Schedule.Wednesday._2nd_Shift_Break1_Length,Break1_Length) ,MOV(LN31_Weekly_Schedule.Wednesday._2nd_Shift_Break2_Length,Break2_Length) ,MOV(LN31_Weekly_Schedule.Wednesday._2nd_Shift_Lunch_Length,Lunch_Length) ,MOV(LN31_Weekly_Schedule.Wednesday.S2_Scheduled,LN31_Schedule.Scheduled_Units) ];
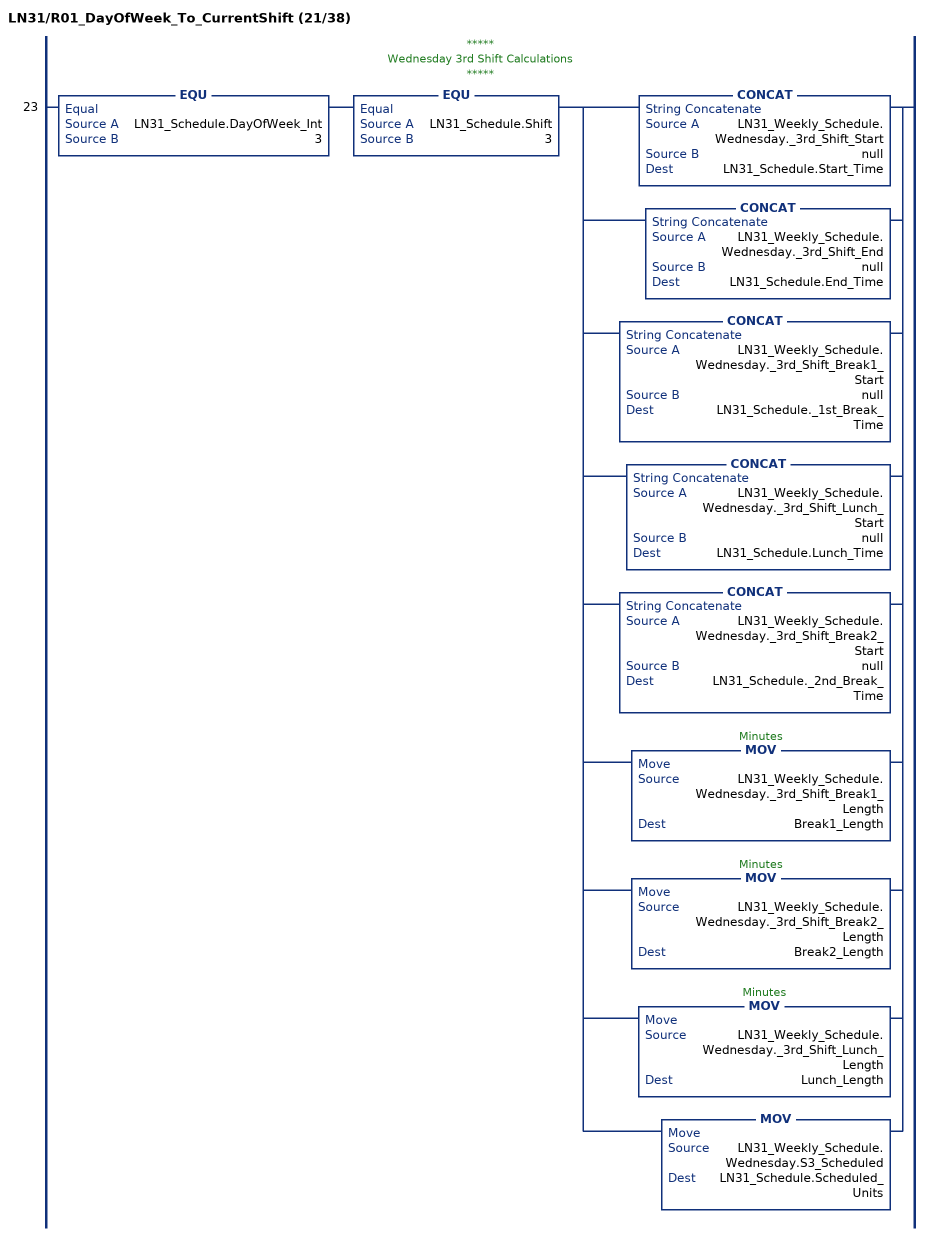
   // *****
   // Wednesday 3rd Shift Calculations
   // *****
   23: EQU(LN31_Schedule.DayOfWeek_Int,3)EQU(LN31_Schedule.Shift,3)[CONCAT(LN31_Weekly_Schedule.Wednesday._3rd_Shift_Start,null,LN31_Schedule.Start_Time) ,CONCAT(LN31_Weekly_Schedule.Wednesday._3rd_Shift_End,null,LN31_Schedule.End_Time) ,CONCAT(LN31_Weekly_Schedule.Wednesday._3rd_Shift_Break1_Start,null,LN31_Schedule._1st_Break_Time) ,CONCAT(LN31_Weekly_Schedule.Wednesday._3rd_Shift_Lunch_Start,null,LN31_Schedule.Lunch_Time) ,CONCAT(LN31_Weekly_Schedule.Wednesday._3rd_Shift_Break2_Start,null,LN31_Schedule._2nd_Break_Time) ,MOV(LN31_Weekly_Schedule.Wednesday._3rd_Shift_Break1_Length,Break1_Length) ,MOV(LN31_Weekly_Schedule.Wednesday._3rd_Shift_Break2_Length,Break2_Length) ,MOV(LN31_Weekly_Schedule.Wednesday._3rd_Shift_Lunch_Length,Lunch_Length) ,MOV(LN31_Weekly_Schedule.Wednesday.S3_Scheduled,LN31_Schedule.Scheduled_Units) ];
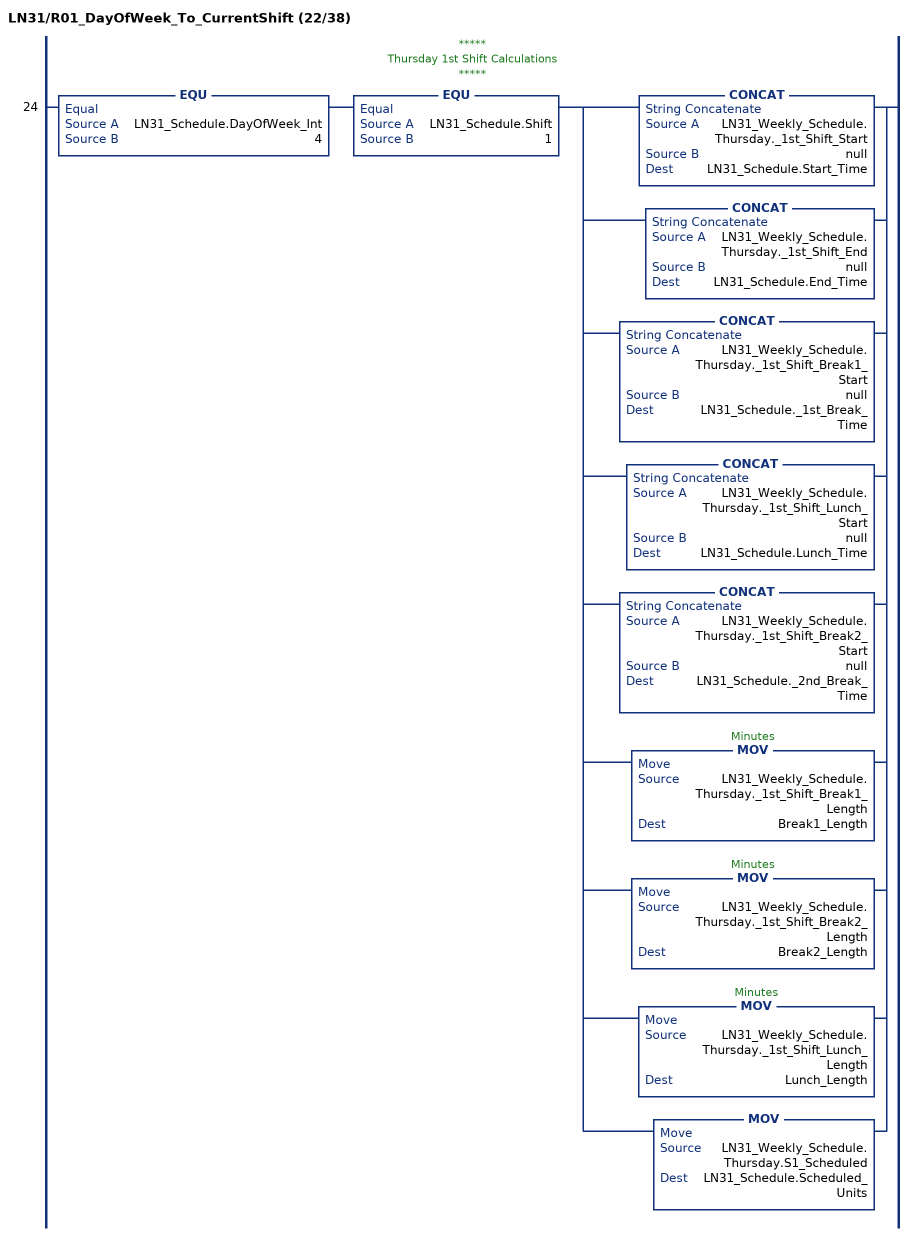
   // *****
   // Thursday 1st Shift Calculations
   // *****
   24: EQU(LN31_Schedule.DayOfWeek_Int,4)EQU(LN31_Schedule.Shift,1)[CONCAT(LN31_Weekly_Schedule.Thursday._1st_Shift_Start,null,LN31_Schedule.Start_Time) ,CONCAT(LN31_Weekly_Schedule.Thursday._1st_Shift_End,null,LN31_Schedule.End_Time) ,CONCAT(LN31_Weekly_Schedule.Thursday._1st_Shift_Break1_Start,null,LN31_Schedule._1st_Break_Time) ,CONCAT(LN31_Weekly_Schedule.Thursday._1st_Shift_Lunch_Start,null,LN31_Schedule.Lunch_Time) ,CONCAT(LN31_Weekly_Schedule.Thursday._1st_Shift_Break2_Start,null,LN31_Schedule._2nd_Break_Time) ,MOV(LN31_Weekly_Schedule.Thursday._1st_Shift_Break1_Length,Break1_Length) ,MOV(LN31_Weekly_Schedule.Thursday._1st_Shift_Break2_Length,Break2_Length) ,MOV(LN31_Weekly_Schedule.Thursday._1st_Shift_Lunch_Length,Lunch_Length) ,MOV(LN31_Weekly_Schedule.Thursday.S1_Scheduled,LN31_Schedule.Scheduled_Units) ];
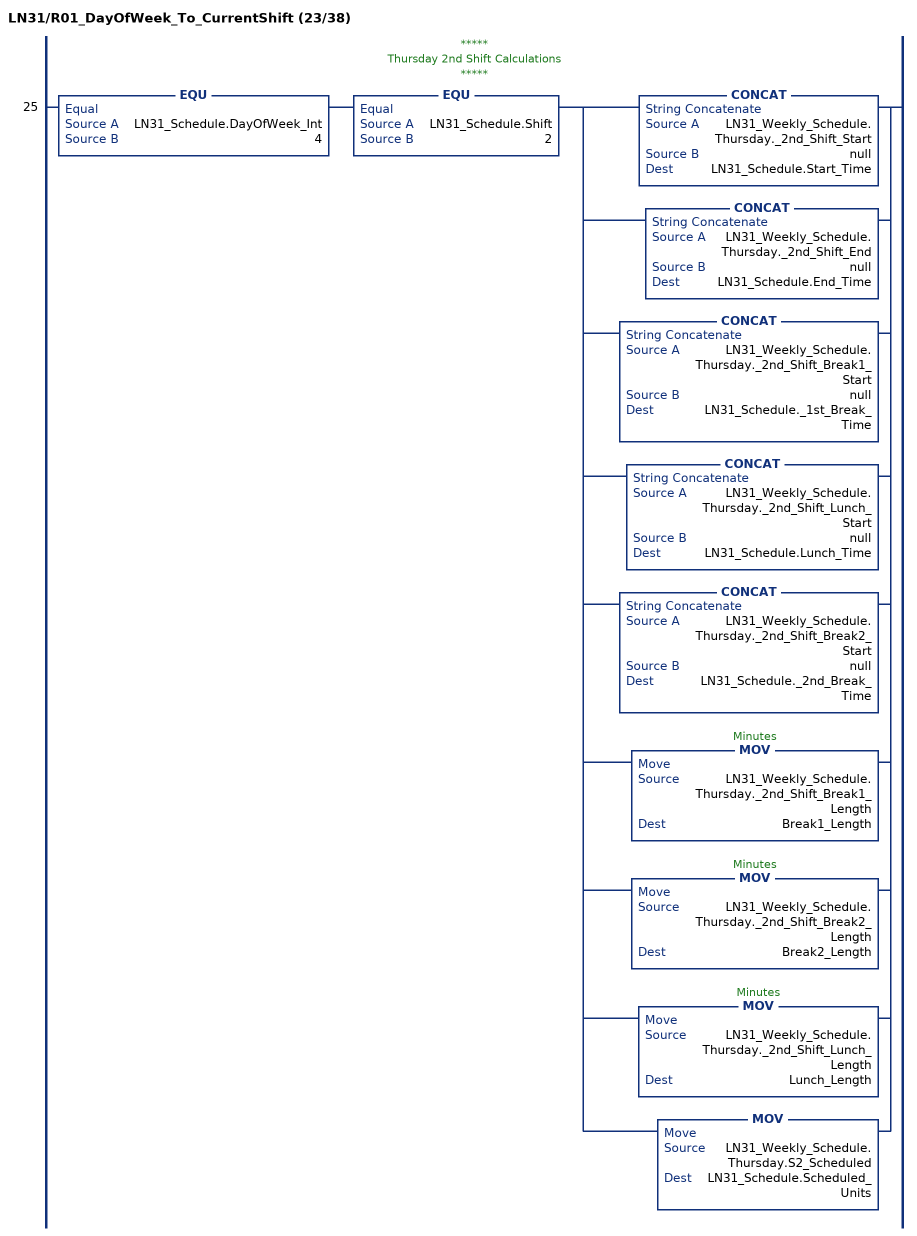
   // *****
   // Thursday 2nd Shift Calculations
   // *****
   25: EQU(LN31_Schedule.DayOfWeek_Int,4)EQU(LN31_Schedule.Shift,2)[CONCAT(LN31_Weekly_Schedule.Thursday._2nd_Shift_Start,null,LN31_Schedule.Start_Time) ,CONCAT(LN31_Weekly_Schedule.Thursday._2nd_Shift_End,null,LN31_Schedule.End_Time) ,CONCAT(LN31_Weekly_Schedule.Thursday._2nd_Shift_Break1_Start,null,LN31_Schedule._1st_Break_Time) ,CONCAT(LN31_Weekly_Schedule.Thursday._2nd_Shift_Lunch_Start,null,LN31_Schedule.Lunch_Time) ,CONCAT(LN31_Weekly_Schedule.Thursday._2nd_Shift_Break2_Start,null,LN31_Schedule._2nd_Break_Time) ,MOV(LN31_Weekly_Schedule.Thursday._2nd_Shift_Break1_Length,Break1_Length) ,MOV(LN31_Weekly_Schedule.Thursday._2nd_Shift_Break2_Length,Break2_Length) ,MOV(LN31_Weekly_Schedule.Thursday._2nd_Shift_Lunch_Length,Lunch_Length) ,MOV(LN31_Weekly_Schedule.Thursday.S2_Scheduled,LN31_Schedule.Scheduled_Units) ];
